	rtM50Ack				: R_TRIG;
	rtM61Ack				: R_TRIG;
	rtM62Ack				: R_TRIG;
	rtM63Ack				: R_TRIG;
	rtM64Ack				: R_TRIG;
	rtM65Ack				: R_TRIG;
	
	F_Ploter: FB_MX2;
	ui_PPodCzestotliwosc: INT;
	b_FP_CCW: BOOL;
	b_FP_CW: BOOL;
	b_FP_Reset: BOOL;
	seq:INT;
	czas:ARRAY[0..100] OF ton;
	R_Pobranie_Kierownica:R_TRIG;

	Zabral: BOOL;
	
	
	
	bZabral: BOOL;
	iStateRunning: INT;
	bServiceMove: BOOL;

END_VAR

VAR CONSTANT
	nAxes	 : WORD:=2;
END_VAR

// Always clear command in active step

// Read input signals
Act_InUpdate();

// ====================================================
// FBs CALL
Act_FBsCall();
// Monitoring
Act_Monitoring();
	
// Error collection
Act_Error();

Act_MovePath(); 

//automat plotera
A_Ploter_Auto();

// SAFETY CALL 
// Tylko komenda Abort dostepna jest niezaleznie od stanu
IF eMachineCommand = E_MachineCommand.eAbort AND eMachineState <> E_MachineState.eAborted THEN
	eMachineState := E_MachineState.eAborting;
END_IF

// Machine mode change over
CASE eMachineMode OF
	
	E_MachineMode.eAutomatic:
		Act_ModeAutomatic();
		
	E_MachineMode.eManual:
		Act_ModeManual();	
		
	E_MachineMode.eMaintenance:
		Act_ModeMaintenance();	
		
END_CASE

// Call Axis online FBs


// Write outputs
Act_OutUpdate(); 
A_FPloter();
A_Prawidlo();

(*//jogi
IF  GVL_HMI.bAuto=FALSE  THEN
	GVL_GLOBAL.bPlotJogF:=GVL_HMI.bHmiPlotCw;
	GVL_GLOBAL.bPlotJogB:=GVL_HMI.bHmiPlotCCw;
END_IF*)

ACTION A_FPloter:
F_Ploter
	(w_Status:=GVL_Omron.wOmron_Pl_Status,
	ui_CzestotliwoscI:=ui_PPodCzestotliwosc,
	b_CCW									:= b_FP_CCW, 
	b_CW									:= b_FP_CW,
	b_Reset                                 := b_FP_Reset,
	w_ControlW                              => GVL_Omron.wOmron_Pl_Control,
 	ui_CzestotliwoscO                       => GVL_Omron.iOmron_Pl_SeVelo,
);

	
	IF GVL_HMI.A_Start=TRUE AND GVL_HMI.bAuto=TRUE AND GVL_HMI.bEnablePloter=TRUE THEN 
		
	ui_PPodCzestotliwosc					:= 2500;
	b_FP_CCW								:= TRUE;		
	
	END_IF	
	IF GVL_HMI.A_Stop=TRUE OR GVL_HMI.bEnablePloter=FALSE THEN  

	b_FP_CCW								:= FALSE;		
	b_FP_CW:=FALSE;
	END_IF
	
	IF GVL_HMI.bAuto=FALSE AND GVL_GLOBAL.falownik_rolek_cewka=TRUE THEN 
	ui_PPodCzestotliwosc					:= 2500;	
	b_FP_CCW								:= TRUE;
	b_FP_CW 								:= FALSE;
	
	
	ELSIF GVL_HMI.bAuto=FALSE AND GVL_GLOBAL.falownik_pasow_cewka=FALSE THEN
	
	ui_PPodCzestotliwosc					:= 0;	
	b_FP_CCW								:= 0;
	b_FP_CW									:= 0;

	END_IF
END_ACTION

ACTION A_Ploter_Auto:
//prędkości osi 
					rItemPickVelocity:=GVL_Recipe.Predk_plot_ruch; 	//[mm/min]
					rItemPlaceVelocity:=GVL_Recipe.Predk_plot_ruch;	//[mm/min]
					rMoveVelocity:=GVL_Recipe.Predk_plot_pobranie;		//[mm/min]
//podglad bitów do obsłgui programu
					R_Pobranie_Kierownica(CLK:=GVL_GLOBAL.Zabierz_Z_Kierownicy);
					R_bReadyForMove(CLK:=bReadyForMove);
				
					bZabral;
					GVL_GLOBAL.odloz_do_kartonu;
//automat do plotera 
				(*	IF GVL_HMI.A_Stop=TRUE OR GVL_HMI.bEnablePloter=FALSE THEN	
					seq									:=0;
					END_IF
				*)	
//rozpoczęcie case
		CASE seq OF 
			0:(*start*)			
					IF GVL_HMI.A_Start=TRUE AND GVL_HMI.bEnablePloter=TRUE THEN	
					seq									:=2;
					END_IF
			2:(*Jazda do home i sprawdzenie stanów *)
					bReferneceHbot						:=TRUE;
					GVL_GLOBAL.zaw_chwyt1_auto			:=FALSE;
					GVL_GLOBAL.zaw_chwyt2_auto			:=FALSE;
					IF GVL_Machine.eState=60 AND bReadyForMove=TRUE AND rMoveMode=3  THEN 
					seq									:=3;
					END_IF
			3:(**)	
					IF bReadyForMove=TRUE AND czas[1].Q=TRUE THEN	
					bMoveCmd							:=TRUE;
					END_IF
					IF bReadyForMove=FALSE THEN	
					bMoveCmd							:=FALSE;
					seq									:=5;
					END_IF
			5:(*sprawdza czy dojechał jak dojechał to jedzie dalej *)
					IF bHome=TRUE THEN
					bHomeDone							:=TRUE;
					seq									:=7;
					END_IF			
			7:(*czeka az zniknie bit bhome*)		
					IF bHome=FALSE THEN
					bHomeDone							:=FALSE;
					seq									:=10;
					END_IF	
			10:(*jade pick pozycje*)
					
					bPickAndPlace						:=TRUE;
					IF rMoveMode=1 AND czas[2].Q=TRUE  THEN
					bPickAndPlace						:=FALSE;
					seq									:=13;
					END_IF
			13:(**)
					IF   bReadyForMove=TRUE THEN
					bMoveCmd							:=TRUE;
					seq									:=14;
					END_IF
			14:(**)	
					IF   bReadyForMove=FALSE THEN
					bMoveCmd							:=FALSE;
					seq									:=15;
					END_IF
			15:(**)	
					IF bReadyToPick=TRUE AND GVL_GLOBAL.Zabierz_Z_Kierownicy  THEN
					bReadyToPickACK						:=TRUE;
					seq									:=17;
					END_IF
			17:(**)	
					IF bReadyToPick=FALSE THEN
					bReadyToPickACK						:=FALSE;
					seq									:=19;						
					END_IF
			19:(**)
				 	IF bPicked=TRUE AND bZabral=TRUE THEN
					GVL_GLOBAL.zaw_chwyt1_auto			:=TRUE;
					GVL_GLOBAL.zaw_chwyt2_auto			:=TRUE;
					seq									:=20;	
					END_IF
					
			20:(*jedzio pobrac jak ma zgode*)

					IF bPicked=TRUE AND czas[4].Q=TRUE THEN
					bPickedACK							:=TRUE;						
					seq									:=22;
					END_IF
			22:(**)		
					IF bPicked=FALSE THEN
					bPickedACK							:=FALSE;						
					seq									:=25;
					END_IF			

					
			25:(*jak zgoda odklada*)
					IF bReadyToPlace=TRUE AND GVL_GLOBAL.odloz_do_kartonu=TRUE THEN
					bReadyToPlaceACK					:=TRUE;
					seq									:=27;
					END_IF

			27:(**)
					IF bReadyToPlace=FALSE   THEN
					bReadyToPlaceACK					:=FALSE;
					seq									:=30;
					END_IF
			30:(*potwierdzenie ze dojechal do pobrania *)
					IF bPlaced	=TRUE  THEN
					GVL_GLOBAL.Ploter_pobral			:=TRUE;
					bPlacedACK							:=TRUE;
					seq									:=33;
					END_IF
			33:(**)		
					IF bPlaced	=FALSE  THEN
					bPlacedACK							:=FALSE;
					seq									:=35;
					END_IF
			35:(*jak zgoda to jedzie spowrotem do pobrania *)
					GVL_GLOBAL.zaw_chwyt1_auto			:=FALSE;
					GVL_GLOBAL.zaw_chwyt2_auto			:=FALSE;
					bReturnToPick						:=TRUE;
					IF rMoveMode = 2  AND czas[3].Q=TRUE  THEN
					seq									:=40;
					END_IF
			40:(**)
					IF bReadyForMove=TRUE THEN
					bMoveCmd							:=TRUE;
					seq									:=43;	
					END_IF
			43:(**)
					IF bReadyForMove=FALSE THEN
					bMoveCmd							:=FALSE;
					seq									:=45;	
					END_IF

			45:(**)
					IF P_HBot_v3.stMcAxisOnline_MCS_X.stStatus.lrActPos<700 THEN 
					GVL_GLOBAL.bZaladowanyPrawidlo		:=TRUE;
					END_IF
					IF bPicked	=TRUE THEN	
					bPickedACK							:=TRUE;
					seq									:=50;//bedzie wracal do 10 
					END_IF
			50:(**)
					IF bPicked	=FALSE THEN	
					bPickedACK							:=FALSE;
					seq									:=10;//bedzie wracal do 10 					
					END_IF
			END_CASE
			czas[1](IN:=seq=3,PT:=T#1200MS);
			czas[2](IN:=rMoveMode=1,PT:=T#1200MS);
			czas[3](IN:=rMoveMode=2,PT:=T#1200MS);
			czas[4](IN:=seq=20,PT:=T#500MS);
			czas[9](IN:=bReferneceHbot,PT:=T#300MS);
			czas[12](IN:=GVL_GLOBAL.bZaladowanyPrawidlo,PT:=T#500MS);

			IF czas[12].Q=TRUE THEN
				GVL_GLOBAL.bZaladowanyPrawidlo	:=FALSE;
			END_IF
END_ACTION

ACTION A_Prawidlo:
FB_Prawidlo(
	b_Start:=GVL_HMI.A_Start AND GVL_HMI.bEnablePloter , 
	b_Stop:=GVL_HMI.A_Stop , 
	bKon_Hamulec1:=GVL_IO_P.b1B1 , 
	bKon_Hamulec2:=GVL_IO_P.b5B1 , 
	bKonPodajnik1:=GVL_IO_P.b6B1 , 
	bKonPodajnik2:=GVL_IO_P.b2B1 , 
	bCzHamulec:=GVL_IO_P.b3B1 , 
	bZaladowany:=GVL_GLOBAL.bZaladowanyPrawidlo	 , 
	bZaworPodnosnik1=>GVL_GLOBAL.zaw_prawidlo_auto , 
	bZaworPodnosnik2=>GVL_GLOBAL.zaw_prawidlo_dol_auto , 
	bZaworHamulec=>GVL_GLOBAL.zaw_hamulec_auto , 
	bZgodaNaRuch=>GVL_GLOBAL.bZgodaNaRuchPrawidlo , 
	bLaduj=>GVL_GLOBAL.odloz_do_kartonu );
END_ACTION

ACTION Act_Error:
// Program summary error
bError := 	tonAxesError.Q OR 
			PLCMachineMode[GVL_NCI.nChan].Error OR  
			PRG_KinTrans.eKinStatus = KinStatus_Error;
			// ie. Init Error
			// OR axis error
			// OR item error
END_ACTION

ACTION Act_FBsCall:

PRG_ChannelHandler();
fbMcAxisOnline_MCS_X(stMcAxisOnline:= stMcAxisOnline_MCS_X , Axis:= Axis_MCS_X);
fbMcAxisOnline_MCS_Y(stMcAxisOnline:= stMcAxisOnline_MCS_y , Axis:= Axis_MCS_Y);
fbMcAxisOnline_ACS_X(stMcAxisOnline:= stMcAxisOnline_ACS_X , Axis:= Axis_ACS_X);
fbMcAxisOnline_ACS_Y(stMcAxisOnline:= stMcAxisOnline_ACS_Y , Axis:= Axis_ACS_Y);	


//________Kinematic____________//
PRG_KinTrans(
	bBuildKinGroup:= , 
	bCleanKinGroup:= , 
	bResetKinGroup:= , 
	bKinBusy=> , 
	bKinDone=> , 
	bKinBuilt=> , 
	bKinClined=> , 
	bKinError=> , 
	udiKinErrorID=> , 
	eKinStatus=> );
//_____________________________//

//________NCI__________________//
PRG_GroupAxesToNci(	stMachineMode := PLCMachineMode[PLCSelectedChannel], 
					stAxisRef_X:= Axis_MCS_X, 
					stAxisRef_Y:= Axis_MCS_Y );

//_____________________________//
END_ACTION

ACTION Act_InUpdate:
bIn1 := TRUE; // Assign, filters, conditions, scaling etc
PLCMachineMode[GVL_NCI.nChan].ProgramName := 'C:\TwinCat\CNC\NC_1.nc';
END_ACTION

ACTION Act_ModeAutomatic:
// State Machine
CASE eMachineState OF

	E_MachineState.eIdle:
		
	
		// ====================================================
		// There should be main code
		// i.e. CASE iStepInit OF	
		// ====================================================
		// Allow for stop only if conditions are true - in this step we can wait without an error

		
		IF TRUE (* condition *) THEN
			eMachineState 						:= E_MachineState.eStopped;
		END_IF
		
		IF bError THEN
			eMachineState 						:= E_MachineState.eError;
		END_IF
		
	E_MachineState.eStopping:
		PLCMachineMode[GVL_NCI.nChan].Start:= FALSE;
		
		CASE iStateStoping OF
			0:
				PLCMachineMode[GVL_NCI.nChan].Stop:= TRUE;
				IF stMcAxisOnline_MCS_X.stStatus.stAxisStatus.NotMoving AND stMcAxisOnline_MCS_Y.stStatus.stAxisStatus.NotMoving THEN
					PLCMachineMode[GVL_NCI.nChan].Stop:= FALSE;
					iStateStoping := iStateStoping + 10;
				ELSIF stMcAxisOnline_MCS_X.stStatus.bNcError OR stMcAxisOnline_MCS_Y.stStatus.bNcError THEN
					iStateStoping := iStateStoping + 20;
				END_IF
			10:
				IF PRG_KinTrans.bKinBuilt THEN
					PRG_KinTrans.bCleanKinGroup := TRUE;
					iStateStoping := iStateStoping + 10;
				ELSE
					iStateStoping := iStateStoping + 20;	
				END_IF
			20:
				IF PRG_KinTrans.bKinDone THEN
					PRG_KinTrans.bCleanKinGroup 		:= FALSE;
					iStateStoping := iStateStoping + 10;
				ELSIF PRG_KinTrans.bKinError THEN
					PRG_KinTrans.bCleanKinGroup 		:= FALSE;
					iStateStoping := iStateStoping + 10;
				END_IF
				
			30:
				PLCMachineMode[GVL_NCI.nChan].Reset:= TRUE;
				IF ItpGetStateInterpreter(arrNCToPLC_NCIChannel_REF[1]) = 1 THEN
					PLCMachineMode[GVL_NCI.nChan].Reset := FALSE;
					iStateStoping := iStateStoping + 10;
				END_IF
			END_CASE
		IF iStateStoping = 40 (* condition *) THEN
			eMachineState 						:= E_MachineState.eStopped;
			iStateStoping 						:= 0;
		END_IF		
	
	E_MachineState.eStopped:
		
		stMcAxisOnline_MCS_X.mcPower.bEnable 			:= FALSE;
		stMcAxisOnline_MCS_X.mcPower.bEnable_Negative 	:= FALSE;
		stMcAxisOnline_MCS_X.mcPower.bEnable_Positive 	:= FALSE;

		stMcAxisOnline_MCS_Y.mcPower.bEnable 			:= FALSE;
		stMcAxisOnline_MCS_Y.mcPower.bEnable_Negative 	:= FALSE;
		stMcAxisOnline_MCS_Y.mcPower.bEnable_Positive 	:= FALSE;
		
		stMcAxisOnline_ACS_X.mcPower.bEnable 			:= FALSE;
		stMcAxisOnline_ACS_X.mcPower.bEnable_Negative 	:= FALSE;
		stMcAxisOnline_ACS_X.mcPower.bEnable_Positive 	:= FALSE;
		
		stMcAxisOnline_ACS_Y.mcPower.bEnable 			:= FALSE;
		stMcAxisOnline_ACS_Y.mcPower.bEnable_Negative 	:= FALSE;
		stMcAxisOnline_ACS_Y.mcPower.bEnable_Positive 	:= FALSE;
	
		
		IF eMachineCommand = E_MachineCommand.eRun THEN
			eMachineState 						:= E_MachineState.eStarting;
		END_IF

		IF eMachineCommand = E_MachineCommand.eRestart THEN
			GVL_Machine.eCommand				:= E_MachineCommand.eStop;
			eMachineState 						:= E_MachineState.eRestarting;
		END_IF			
				
		IF bError THEN
			eMachineState 						:= E_MachineState.eError;
		END_IF

	E_MachineState.eStarting:
		PLCMachineMode[GVL_NCI.nChan].Manual 	:= FALSE;

		CASE iStepStarting OF
			0:
				PLCMachineMode[GVL_NCI.nChan].Stop				:= FALSE;
				
				stMcAxisOnline_MCS_X.mcPower.bEnable 			:= TRUE;
				stMcAxisOnline_MCS_X.mcPower.bEnable_Negative 	:= TRUE;
				stMcAxisOnline_MCS_X.mcPower.bEnable_Positive 	:= TRUE;
				stMcAxisOnline_MCS_X.mcPower.lrOverride		 	:= 100.0;	
	
				stMcAxisOnline_MCS_Y.mcPower.bEnable 			:= TRUE;
				stMcAxisOnline_MCS_Y.mcPower.bEnable_Negative 	:= TRUE;
				stMcAxisOnline_MCS_Y.mcPower.bEnable_Positive 	:= TRUE;
				stMcAxisOnline_MCS_Y.mcPower.lrOverride		 	:= 100.0;	
				
				stMcAxisOnline_ACS_X.mcPower.bEnable 			:= TRUE;
				stMcAxisOnline_ACS_X.mcPower.bEnable_Negative 	:= TRUE;
				stMcAxisOnline_ACS_X.mcPower.bEnable_Positive 	:= TRUE;
				stMcAxisOnline_ACS_X.mcPower.lrOverride		 	:= 100.0;	
				
				stMcAxisOnline_ACS_Y.mcPower.bEnable 			:= TRUE;
				stMcAxisOnline_ACS_Y.mcPower.bEnable_Negative 	:= TRUE;
				stMcAxisOnline_ACS_Y.mcPower.bEnable_Positive 	:= TRUE;
				stMcAxisOnline_ACS_Y.mcPower.lrOverride		 	:= 100.0;	
				
				IF tonAxesReady.Q THEN
					iStepStarting := iStepStarting + 10;
				ELSIF tonAxesError.Q THEN
					bError := TRUE;
				END_IF
			10:
				PLCMachineMode[GVL_NCI.nChan].Automatic := TRUE;
				IF PLCNciChannelState.Mode[GVL_NCI.nChan] = 2 THEN
					iStepStarting := iStepStarting + 10;
				END_IF
			20:
			
				IF PRG_KinTrans.bKinBuilt AND NOT PRG_KinTrans.bKinError THEN
					iStepStarting := iStepStarting + 20;		
				ELSE
					iStepStarting := iStepStarting + 10;
				END_IF
				
			30:
				PRG_KinTrans.bBuildKinGroup := TRUE;
					IF PRG_KinTrans.bKinDone THEN
						PRG_KinTrans.bBuildKinGroup := FALSE;
						iStepStarting := iStepStarting + 10;
					END_IF
			40:
				;
			END_CASE 
	
		IF iStepStarting = 40 AND PRG_KinTrans.eKinStatus = KinStatus_Ready(* condition *) THEN
			eMachineState 						:= E_MachineState.eRunning;
			iStepStarting 						:= 0;
		END_IF
		
	E_MachineState.eRunning:
		
		//Act_MovePath();  do usuniecia
		PLCMachineMode[GVL_NCI.nChan].Start 	:= GVL_Machine.bNciStart;
		PLCMachineMode[GVL_NCI.nChan].Stop 		:= GVL_Machine.bNCiStop;
	
		GVL_Machine.bNciFeedHold := ItpIsEStopEx(arrNCToPLC_NCIChannel_REF[1]);
		
		// ====================================================
		// There should be main code
		// i.e. CASE iStepAuto OF
		// ====================================================
		IF eMachineCommand = E_MachineCommand.eStop OR bError THEN
			eMachineState 						:= E_MachineState.eStopping;
		END_IF

	E_MachineState.eAborting:

		// Stop and reset everything - usually SAFETY function
		CASE iStateAborting OF
			0:
				IF ItpGetStateInterpreter(arrNCToPLC_NCIChannel_REF[1]) <> 1 THEN
					iStateAborting := iStateAborting +10;
				ELSE
					iStateAborting := iStateAborting + 20;
				END_IF
			10:
				PLCMachineMode[GVL_NCI.nChan].Stop:= TRUE;
					IF ItpIsEStopEx(arrNCToPLC_NCIChannel_REF[1]) THEN
						PLCMachineMode[GVL_NCI.nChan].Stop:= FALSE;
						iStateAborting := iStateAborting +10;
					ELSIF 	ItpGetStateInterpreter(arrNCToPLC_NCIChannel_REF[1]) <> 1 OR
							ItpGetStateInterpreter(arrNCToPLC_NCIChannel_REF[1]) <> 12 OR
							ItpGetStateInterpreter(arrNCToPLC_NCIChannel_REF[1]) <> 13 THEN
						PLCMachineMode[GVL_NCI.nChan].Stop:= FALSE;
						iStateAborting := iStateAborting +10;
					END_IF
			20:
				IF PRG_KinTrans.bKinBuilt THEN
					PRG_KinTrans.bCleanKinGroup := TRUE;
					iStateAborting := iStateAborting + 10;
				ELSE	
					iStateAborting := iStateAborting + 20;
				END_IF
			30:
				IF PRG_KinTrans.bKinDone THEN
					PRG_KinTrans.bCleanKinGroup := FALSE;
					iStateAborting := iStateAborting + 10;
				ELSIF PRG_KinTrans.bKinError THEN
					PRG_KinTrans.bCleanKinGroup := FALSE;
					iStateAborting := iStateAborting + 10;
				END_IF
			40:	
				PLCMachineMode[GVL_NCI.nChan].Manual := TRUE;
				stMcAxisOnline_ACS_X.mcSS1.bExecute := TRUE;
				stMcAxisOnline_ACS_Y.mcSS1.bExecute := TRUE;
				IF stMcAxisOnline_ACS_X.mcSS1.bDone AND stMcAxisOnline_ACS_Y.mcSS1.bDone THEN
					iStateAborting := iStateAborting + 10;
				ELSIF stMcAxisOnline_ACS_X.mcSS1.bError OR stMcAxisOnline_ACS_Y.mcSS1.bError THEN
					iStateAborting := iStateAborting + 10;
				END_IF
			50:	

				stMcAxisOnline_MCS_X.mcSS1.bExecute := Axis_MCS_X.Status.PTPmode;
				stMcAxisOnline_MCS_Y.mcSS1.bExecute := Axis_MCS_Y.Status.PTPmode;
			
				IF 	stMcAxisOnline_MCS_X.mcSS1.bDone AND stMcAxisOnline_MCS_Y.mcSS1.bDone THEN
					iStateAborting := iStateAborting + 10;
				ELSIF stMcAxisOnline_MCS_X.mcSS1.bError OR stMcAxisOnline_MCS_Y.mcSS1.bError THEN
					iStateAborting := iStateAborting + 10;
				END_IF	
			
			60:
				stMcAxisOnline_MCS_X.mcSS1.bExecute := TRUE;
				stMcAxisOnline_MCS_Y.mcSS1.bExecute := TRUE;
				stMcAxisOnline_ACS_X.mcSS1.bExecute := TRUE;;
				stMcAxisOnline_ACS_Y.mcSS1.bExecute := TRUE;
		END_CASE
	
		IF iStateAborting = 60 THEN
			eMachineState 						:= E_MachineState.eAborted;
			iStateAborting						:= 0;
		END_IF		
		
	E_MachineState.eAborted:

		stMcAxisOnline_MCS_X.mcSS1.bExecute := NOT GVL_SafetyFrom_RT2.bSAFETY_PermissionSS1;
		stMcAxisOnline_MCS_Y.mcSS1.bExecute := NOT GVL_SafetyFrom_RT2.bSAFETY_PermissionSS1;
		stMcAxisOnline_ACS_X.mcSS1.bExecute := NOT GVL_SafetyFrom_RT2.bSAFETY_PermissionSS1;
		stMcAxisOnline_ACS_Y.mcSS1.bExecute := NOT GVL_SafetyFrom_RT2.bSAFETY_PermissionSS1;
					
		IF eMachineCommand = E_MachineCommand.eReset THEN
			eMachineState 						:= E_MachineState.eReseting;
		END_IF
		
		IF bError THEN
			eMachineState 						:= E_MachineState.eError;
		END_IF

	E_MachineState.eError:

		// ====================================================
		// Two types of error:
		// 1. 'Small/soft' Error - fix a problem and go to stop
		// 2. 'Serious/hard' Error - there is a need of restart everything, if there is a sequence - reset it too - fix a problem and go to init
		// ====================================================
		stMcAxisOnline_MCS_X.mcReset.bExecute	:= FALSE;	
		stMcAxisOnline_MCS_Y.mcReset.bExecute 	:= FALSE;	
		stMcAxisOnline_ACS_X.mcReset.bExecute 	:= FALSE;	
		stMcAxisOnline_ACS_Y.mcReset.bExecute 	:= FALSE;	
		stMcAxisOnline_MCS_X.mcStop.bExecute 	:= FALSE;
		stMcAxisOnline_MCS_Y.mcStop.bExecute	:= FALSE;
		stMcAxisOnline_ACS_X.mcStop.bExecute 	:= FALSE;
		stMcAxisOnline_ACS_Y.mcStop.bExecute	:= FALSE;
		PRG_KinTrans.bResetKinGroup 			:= FALSE;
		PRG_KinTrans.bBuildKinGroup 			:= FALSE;
		PRG_KinTrans.bCleanKinGroup 			:= FALSE;		
		PLCMachineMode[GVL_NCI.nChan].Reset 	:= FALSE;		
		PLCMachineMode[GVL_NCI.nChan].Stop		:= FALSE;
		PLCMachineMode[GVL_NCI.nChan].Start		:= FALSE;
	
		IF eMachineCommand = E_MachineCommand.eReset THEN
			eMachineState 						:= E_MachineState.eReseting;
		END_IF
		
		IF eMachineCommand = E_MachineCommand.eRestart THEN
			eMachineState 						:= E_MachineState.eRestarting;
		END_IF

	E_MachineState.eReseting:

		// ====================================================
		//'Small/soft' Error - fix a problem and go to stop
		// Reset drives only when it is necessary
		// ====================================================
		// Check if axis errors cleared
	
		IF PRG_KinTrans.eKinStatus = KinStatus_Error OR PRG_KinTrans.bKinError	THEN
			PRG_KinTrans.bResetKinGroup := TRUE;
		ELSIF PLCMachineMode[GVL_NCI.nChan].Error THEN
			PLCMachineMode[GVL_NCI.nChan].Reset := TRUE;
		ELSIF stMcAxisOnline_MCS_X.stError.bError THEN
			stMcAxisOnline_MCS_X.mcReset.bExecute := TRUE;
		ELSIF stMcAxisOnline_MCS_Y.stError.bError THEN
			stMcAxisOnline_MCS_Y.mcReset.bExecute := TRUE;	
		ELSIF stMcAxisOnline_ACS_X.stError.bError THEN
			stMcAxisOnline_ACS_X.mcReset.bExecute := TRUE;
		ELSIF stMcAxisOnline_ACS_Y.stError.bError THEN
			stMcAxisOnline_ACS_Y.mcReset.bExecute := TRUE;
		END_IF

	
		IF NOT tonAxesError.Q AND NOT PLCMachineMode[GVL_NCI.nChan].Error AND PRG_KinTrans.eKinStatus <> KinStatus_Error AND NOT PRG_KinTrans.bKinError THEN
			stMcAxisOnline_MCS_X.mcReset.bExecute	:= FALSE;	
			stMcAxisOnline_MCS_Y.mcReset.bExecute 	:= FALSE;	
			stMcAxisOnline_ACS_X.mcReset.bExecute 	:= FALSE;	
			stMcAxisOnline_ACS_Y.mcReset.bExecute 	:= FALSE;	
			PRG_KinTrans.bResetKinGroup 			:= FALSE;
			PLCMachineMode[GVL_NCI.nChan].Reset		:= FALSE;
			eMachineState  						:= E_MachineState.eStopping;
		END_IF
				
		// Blad bloku resetowania lub zakonczylismy kasowanie bledu osi, ale os jest nadal w bledzie, np. nie usunieta usterka - idz do kroku bledu
		IF bError (*(stAxis.stAxisDiagOutputs.Error OR (stAxis.stAxisDiagOutputs.Done AND stAxis.bAxisError)) *) THEN
			eMachineState  						:= E_MachineState.eError;
		END_IF
		
	E_MachineState.eRestarting:

		// ====================================================
		// 'Serious/hard' Error - there is a need of restart everything, if there is a sequence - reset it too - fix a problem and go to init
		// Reset drives only when it is necessary
		// ====================================================
		// Check if axis errors cleared
		bError := FALSE;
		
		IF TRUE (*NOT bAxisError AND NOT other errors *) THEN
			eMachineState  						:= E_MachineState.eIdle;
		END_IF
				
		// Blad bloku resetowania lub zakonczylismy kasowanie bledu osi, ale os jest nadal w bledzie, np. nie usunieta usterka - idz do kroku bledu
		IF bError (*(stAxis.stAxisDiagOutputs.Error OR (stAxis.stAxisDiagOutputs.Done AND stAxis.bAxisError)) *) THEN
			eMachineState  						:= E_MachineState.eError;
		END_IF
		
END_CASE
END_ACTION

ACTION Act_ModeMaintenance:
// State Machine
CASE eMachineState OF

	E_MachineState.eIdle, E_MachineState.eStopping, E_MachineState.eStopped, E_MachineState.eStarting:
	
		// ====================================================
		// There should be main code
		// i.e. CASE iStepInit OF	
		// ====================================================
		// Allow for stop only if conditions are true - in this step we can wait without an error	
		IF TRUE (* condition *) AND eMachineCommand = E_MachineCommand.eRun THEN
			eMachineState 						:= E_MachineState.eRunning;
		END_IF

	E_MachineState.eRunning:

		// ====================================================
		// HMI control
		// There should be main code,
		// i.e. CASE iStepAuto OF
		// ====================================================
		IF eMachineCommand = E_MachineCommand.eStop THEN
			eMachineState 						:= E_MachineState.eStopping;
		END_IF

	E_MachineState.eAborting:

		// Stop and reset everything - usually SAFETY function
		IF TRUE (* condition *) THEN
			eMachineState 						:= E_MachineState.eAborted;
		END_IF
		
	E_MachineState.eAborted:

		IF eMachineCommand = E_MachineCommand.eReset THEN
			eMachineState 						:= E_MachineState.eReseting;
		END_IF

	E_MachineState.eRestarting, E_MachineState.eReseting, E_MachineState.eError:

			;// Unused

END_CASE
END_ACTION

ACTION Act_ModeManual:
// State Machine

CASE eMachineState OF

	E_MachineState.eIdle:
	
		// ====================================================
		// There should be main code
		// i.e. CASE iStepInit OF	
		// ====================================================
		// Allow for stop only if conditions are true - in this step we can wait without an error

		CASE iStateIdle OF
			0:	//Wyłączenie kanału interpolacji
				PLCMachineMode[GVL_NCI.nChan].Automatic 		:= FALSE;
				PLCMachineMode[GVL_NCI.nChan].Manual			:= TRUE;
				IF arrNCToPLC_NCIChannel_REF[1].ItpState = 1 THEN
					iStateIdle := iStateIdle + 10;
				END_IF
			10:	
				IF PRG_KinTrans.bKinBuilt THEN
					PRG_KinTrans.bCleanKinGroup := TRUE;
					iStateIdle := iStateIdle + 10;
				ELSE
					iStateIdle := iStateIdle + 20;	
				END_IF
			20:
				IF PRG_KinTrans.bKinDone THEN
					PRG_KinTrans.bCleanKinGroup 		:= FALSE;
					iStateIdle := iStateIdle + 10;
				ELSIF PRG_KinTrans.bKinError THEN
					PRG_KinTrans.bCleanKinGroup 		:= FALSE;
					iStateIdle := iStateIdle + 10;
				END_IF
			END_CASE
	
		IF iStateIdle = 30 (* condition *)THEN
			eMachineState 						:= E_MachineState.eStopped;
			iStateIdle							:= 0;		
		END_IF
		
		IF bError THEN
			eMachineState 						:= E_MachineState.eError;
			iStateIdle							:= 0;	
		END_IF

	E_MachineState.eStopping:	
		CASE iStateStoping OF
			0:	

				stMcAxisOnline_MCS_X.mcStop.bExecute := TRUE;
				stMcAxisOnline_MCS_Y.mcStop.bExecute := TRUE;
				IF 	stMcAxisOnline_MCS_X.mcStop.bDone AND stMcAxisOnline_MCS_Y.mcStop.bDone THEN
					iStateStoping := iStateStoping + 10;
				ELSIF stMcAxisOnline_MCS_X.mcStop.bError OR stMcAxisOnline_MCS_Y.mcStop.bError THEN
					iStateStoping := iStateStoping + 10;
				END_IF	
			10:
				stMcAxisOnline_MCS_X.mcStop.bExecute := FALSE;
				stMcAxisOnline_MCS_Y.mcStop.bExecute := FALSE;
				iStateStoping := iStateStoping + 10;
			20:
				PRG_KinTrans.bCleanKinGroup := TRUE;
				IF PRG_KinTrans.bKinDone THEN
					PRG_KinTrans.bCleanKinGroup 		:= FALSE;
					iStateStoping := iStateStoping + 10;
				END_IF	
		END_CASE
		
		IF iStateStoping = 30 (* condition *) THEN
			eMachineState 						:= E_MachineState.eStopped;
			iStateStoping 						:= 0;
		END_IF			
	
		IF bError THEN
			eMachineState 						:= E_MachineState.eError;
		END_IF		
	
	E_MachineState.eStopped:
			
				stMcAxisOnline_MCS_X.mcPower.bEnable 			:= FALSE;
				stMcAxisOnline_MCS_X.mcPower.bEnable_Negative 	:= FALSE;
				stMcAxisOnline_MCS_X.mcPower.bEnable_Positive 	:= FALSE;
		
				stMcAxisOnline_MCS_Y.mcPower.bEnable 			:= FALSE;
				stMcAxisOnline_MCS_Y.mcPower.bEnable_Negative 	:= FALSE;
				stMcAxisOnline_MCS_Y.mcPower.bEnable_Positive 	:= FALSE;
				
				stMcAxisOnline_ACS_X.mcPower.bEnable 			:= FALSE;
				stMcAxisOnline_ACS_X.mcPower.bEnable_Negative 	:= FALSE;
				stMcAxisOnline_ACS_X.mcPower.bEnable_Positive 	:= FALSE;
				
				stMcAxisOnline_ACS_Y.mcPower.bEnable 			:= FALSE;
				stMcAxisOnline_ACS_Y.mcPower.bEnable_Negative 	:= FALSE;
				stMcAxisOnline_ACS_Y.mcPower.bEnable_Positive 	:= FALSE;
		IF eMachineCommand = E_MachineCommand.eRun THEN
			eMachineState 						:= E_MachineState.eStarting;
		END_IF	

		IF eMachineCommand = E_MachineCommand.eRestart THEN
			GVL_Machine.eCommand				:= E_MachineCommand.eStop;
			eMachineState 						:= E_MachineState.eRestarting;
		END_IF			
		
 	E_MachineState.eStarting:
		CASE iStepStarting OF
			0:
				stMcAxisOnline_MCS_X.mcPower.bEnable 			:= TRUE;
				stMcAxisOnline_MCS_X.mcPower.bEnable_Negative 	:= TRUE;
				stMcAxisOnline_MCS_X.mcPower.bEnable_Positive 	:= TRUE;
				stMcAxisOnline_MCS_X.mcPower.lrOverride		 	:= 100.0;	
			
				stMcAxisOnline_MCS_Y.mcPower.bEnable 			:= TRUE;
				stMcAxisOnline_MCS_Y.mcPower.bEnable_Negative 	:= TRUE;
				stMcAxisOnline_MCS_Y.mcPower.bEnable_Positive 	:= TRUE;
				stMcAxisOnline_MCS_Y.mcPower.lrOverride		 	:= 100.0;	
				
				stMcAxisOnline_ACS_X.mcPower.bEnable 			:= TRUE;
				stMcAxisOnline_ACS_X.mcPower.bEnable_Negative 	:= TRUE;
				stMcAxisOnline_ACS_X.mcPower.bEnable_Positive 	:= TRUE;
				stMcAxisOnline_ACS_X.mcPower.lrOverride		 	:= 100.0;	
				
				stMcAxisOnline_ACS_Y.mcPower.bEnable 			:= TRUE;
				stMcAxisOnline_ACS_Y.mcPower.bEnable_Negative 	:= TRUE;
				stMcAxisOnline_ACS_Y.mcPower.bEnable_Positive 	:= TRUE;
				stMcAxisOnline_ACS_Y.mcPower.lrOverride		 	:= 100.0;	
				IF tonAxesReady.Q THEN
					iStepStarting := iStepStarting + 10;
				END_IF
			10:
				IF PRG_KinTrans.bKinBuilt THEN
					iStepStarting := iStepStarting + 20;
				ELSE
					PRG_KinTrans.bBuildKinGroup := TRUE;
					iStepStarting := iStepStarting + 10;
				END_IF

			20:	
				IF PRG_KinTrans.bKinDone THEN
					PRG_KinTrans.bBuildKinGroup := FALSE;	
					iStepStarting := iStepStarting + 10;
				END_IF
			30:
				;	
		END_CASE
	
		IF iStepStarting = 30 THEN
			eMachineState 						:= E_MachineState.eRunning;
			iStepStarting 						:= 0;
		END_IF
				

		
		IF bError THEN
			eMachineState 							:= E_MachineState.eError;		
			iStepStarting							:= 0;			
		END_IF
	
		
		
	E_MachineState.eRunning:

		// ====================================================
		// HMI control
		// There should be main code,
		// i.e. CASE iStepAuto OF
		// ====================================================
		CASE iStateRunning OF
			0:
				stMcAxisOnline_MCS_Y.mcMoveAbsolute.bExecute := FALSE;
				stMcAxisOnline_MCS_X.mcMoveAbsolute.bExecute := FALSE;
				IF bServiceMove THEN
					bServiceMove := FALSE;
					iStateRunning := iStateRunning + 10;
				END_IF
			10:
				stMcAxisOnline_MCS_Y.mcMoveAbsolute.lrPosition :=  0; //Pozycja
				stMcAxisOnline_MCS_Y.mcMoveAbsolute.lrVelocity :=  10;      //Predkosc
				stMcAxisOnline_MCS_Y.mcMoveAbsolute.bExecute := TRUE;
				IF stMcAxisOnline_MCS_Y.mcMoveAbsolute.bDone THEN
					stMcAxisOnline_MCS_Y.mcMoveAbsolute.bExecute := FALSE;
					iStateRunning := iStateRunning + 10;
				END_IF
			20:
				
				stMcAxisOnline_MCS_X.mcMoveAbsolute.lrPosition :=  0; //Pozycja
				stMcAxisOnline_MCS_X.mcMoveAbsolute.lrVelocity :=  10;      //Predkosc
				stMcAxisOnline_MCS_X.mcMoveAbsolute.bExecute := TRUE;
				IF stMcAxisOnline_MCS_X.mcMoveAbsolute.bDone THEN
					stMcAxisOnline_MCS_X.mcMoveAbsolute.bExecute := FALSE;
					iStateRunning := iStateRunning + 10;
				END_IF
			30:
				;//Dummy wait
			
		END_CASE
		IF eMachineCommand = E_MachineCommand.eStop OR bError THEN
			eMachineState 						:= E_MachineState.eStopping;
			iStateRunning := 0;
		END_IF

	E_MachineState.eAborting:
		CASE iStateAborting OF
			0:
				PLCMachineMode[GVL_NCI.nChan].Automatic 		:= FALSE;
				PLCMachineMode[GVL_NCI.nChan].Manual	 		:= TRUE;
				iStateAborting := iStateAborting + 10;
			10:
				IF PRG_KinTrans.bKinBuilt THEN
					PRG_KinTrans.bCleanKinGroup := TRUE;
					iStateAborting := iStateAborting + 10;
				ELSE	
					iStateAborting := iStateAborting + 20;
				END_IF
			20:
				IF PRG_KinTrans.bKinDone THEN
					PRG_KinTrans.bCleanKinGroup := FALSE;
					iStateAborting := iStateAborting + 10;
				ELSIF PRG_KinTrans.bKinError THEN
					PRG_KinTrans.bCleanKinGroup := FALSE;
					iStateAborting := iStateAborting + 10;
				END_IF
			30:
				stMcAxisOnline_ACS_X.mcSS1.bExecute := TRUE;
				stMcAxisOnline_ACS_Y.mcSS1.bExecute := TRUE;
				
				IF stMcAxisOnline_ACS_X.mcSS1.bDone AND stMcAxisOnline_ACS_Y.mcSS1.bDone THEN
					iStateAborting := iStateAborting + 10;
				ELSIF stMcAxisOnline_ACS_X.mcSS1.bError OR stMcAxisOnline_ACS_Y.mcSS1.bError THEN
					iStateAborting := iStateAborting + 10;
				END_IF	
			40:
				stMcAxisOnline_MCS_X.mcSS1.bExecute := Axis_MCS_X.Status.PTPmode;
				stMcAxisOnline_MCS_Y.mcSS1.bExecute := Axis_MCS_Y.Status.PTPmode;
				IF 	stMcAxisOnline_MCS_X.mcSS1.bDone AND stMcAxisOnline_MCS_Y.mcSS1.bDone THEN
					iStateAborting := iStateAborting + 10;
				ELSIF stMcAxisOnline_MCS_X.mcSS1.bError OR stMcAxisOnline_MCS_Y.mcSS1.bError THEN
					iStateAborting := iStateAborting + 10;
				END_IF	
			50:
				stMcAxisOnline_MCS_X.mcSS1.bExecute := TRUE;
				stMcAxisOnline_MCS_Y.mcSS1.bExecute := TRUE;
				stMcAxisOnline_ACS_X.mcSS1.bExecute := TRUE;
				stMcAxisOnline_ACS_Y.mcSS1.bExecute := TRUE;
				eMachineState 						:= E_MachineState.eAborted;	
		END_CASE
		// Stop and reset everything - usually SAFETY function
		IF iStateAborting = 50 (* condition *) THEN
			eMachineState 						:= E_MachineState.eAborted;
			iStateAborting := 0;
		END_IF
		
	E_MachineState.eAborted:
	
		stMcAxisOnline_MCS_X.mcSS1.bExecute := NOT GVL_SafetyFrom_RT2.bSAFETY_PermissionSS1;
		stMcAxisOnline_MCS_Y.mcSS1.bExecute := NOT GVL_SafetyFrom_RT2.bSAFETY_PermissionSS1;
		stMcAxisOnline_ACS_X.mcSS1.bExecute := NOT GVL_SafetyFrom_RT2.bSAFETY_PermissionSS1;
		stMcAxisOnline_ACS_Y.mcSS1.bExecute := NOT GVL_SafetyFrom_RT2.bSAFETY_PermissionSS1;
		IF eMachineCommand = E_MachineCommand.eReset THEN
			eMachineState 						:= E_MachineState.eReseting;
		END_IF

	E_MachineState.eError:

		// ====================================================
		// Two types of error:
		// 1. 'Small/soft' Error - fix a problem and go to stop
		// 2. 'Serious/hard' Error - there is a need of restart everything, if there is a sequence - reset it too - fix a problem and go to init
		// ====================================================
		stMcAxisOnline_MCS_X.mcReset.bExecute	:= FALSE;	
		stMcAxisOnline_MCS_Y.mcReset.bExecute 	:= FALSE;	
		stMcAxisOnline_ACS_X.mcReset.bExecute 	:= FALSE;	
		stMcAxisOnline_ACS_Y.mcReset.bExecute 	:= FALSE;	
		stMcAxisOnline_MCS_X.mcStop.bExecute 	:= FALSE;
		stMcAxisOnline_MCS_Y.mcStop.bExecute	:= FALSE;
		stMcAxisOnline_ACS_X.mcStop.bExecute 	:= FALSE;
		stMcAxisOnline_ACS_Y.mcStop.bExecute	:= FALSE;
		PRG_KinTrans.bResetKinGroup 			:= FALSE;
		PRG_KinTrans.bBuildKinGroup 			:= FALSE;	
		PRG_KinTrans.bCleanKinGroup 			:= FALSE;		
	
		IF eMachineCommand = E_MachineCommand.eReset THEN
			eMachineState 						:= E_MachineState.eReseting;
		END_IF
		
		IF eMachineCommand = E_MachineCommand.eRestart THEN
			eMachineState 						:= E_MachineState.eRestarting;
		END_IF		
			
		
	E_MachineState.eRestarting, E_MachineState.eReseting:
	
		IF PRG_KinTrans.eKinStatus = KinStatus_Error	THEN
			PRG_KinTrans.bResetKinGroup := TRUE;
		ELSIF PLCMachineMode[GVL_NCI.nChan].Error THEN
			PLCMachineMode[GVL_NCI.nChan].Reset := TRUE;
		ELSIF stMcAxisOnline_MCS_X.stError.bError THEN
			stMcAxisOnline_MCS_X.mcReset.bExecute := TRUE;
		ELSIF stMcAxisOnline_MCS_Y.stError.bError THEN
			stMcAxisOnline_MCS_Y.mcReset.bExecute := TRUE;	
		ELSIF stMcAxisOnline_ACS_X.stError.bError THEN
			stMcAxisOnline_ACS_X.mcReset.bExecute := TRUE;
		ELSIF stMcAxisOnline_ACS_Y.stError.bError THEN
			stMcAxisOnline_ACS_Y.mcReset.bExecute := TRUE;
		END_IF	
	
		IF NOT tonAxesError.Q AND NOT PLCMachineMode[GVL_NCI.nChan].Error AND PRG_KinTrans.eKinStatus <> KinStatus_Error THEN
			stMcAxisOnline_MCS_X.mcReset.bExecute	:= FALSE;	
			stMcAxisOnline_MCS_Y.mcReset.bExecute 	:= FALSE;	
			stMcAxisOnline_ACS_X.mcReset.bExecute 	:= FALSE;	
			stMcAxisOnline_ACS_Y.mcReset.bExecute 	:= FALSE;	
			PRG_KinTrans.bResetKinGroup 			:= FALSE;
			PLCMachineMode[GVL_NCI.nChan].Reset		:= FALSE;
			
			IF eMachineState = E_MachineState.eReseting THEN
				eMachineState  						:= E_MachineState.eStopping;
			END_IF
			
			IF eMachineState = E_MachineState.eRestarting THEN
				eMachineState  						:= E_MachineState.eIdle;	
			END_IF
		END_IF	
	(*
		// Blad bloku resetowania lub zakonczylismy kasowanie bledu osi, ale os jest nadal w bledzie, np. nie usunieta usterka - idz do kroku bledu
		IF bError (*(stAxis.stAxisDiagOutputs.Error OR (stAxis.stAxisDiagOutputs.Done AND stAxis.bAxisError)) *) THEN
			eMachineState  						:= E_MachineState.eError;
		END_IF
			;// Unused
	*)
END_CASE
END_ACTION

ACTION Act_Monitoring:
// Ustawianie flag, monitoring kolizjii, watchdogi, jazdy po krzywce itp
tonAxesReady.IN := 	stMcAxisOnline_ACS_X.mcPower.bStatus AND stMcAxisOnline_ACS_X.stStatus.bAxisReady AND
					stMcAxisOnline_ACS_Y.mcPower.bStatus AND stMcAxisOnline_ACS_Y.stStatus.bAxisReady AND
					stMcAxisOnline_MCS_X.mcPower.bStatus AND stMcAxisOnline_MCS_X.stStatus.bAxisReady AND
					stMcAxisOnline_MCS_Y.mcPower.bStatus AND stMcAxisOnline_MCS_Y.stStatus.bAxisReady	;
tonAxesReady(PT:=T#200MS);

tonAxesError.IN := 	stMcAxisOnline_ACS_X.stError.bDriveError OR stMcAxisOnline_ACS_X.stError.bNcError OR
					stMcAxisOnline_ACS_Y.stError.bDriveError OR stMcAxisOnline_ACS_Y.stError.bNcError OR
					stMcAxisOnline_MCS_X.stError.bDriveError OR stMcAxisOnline_MCS_X.stError.bNcError OR
					stMcAxisOnline_MCS_Y.stError.bDriveError OR stMcAxisOnline_MCS_Y.stError.bNcError	;
tonAxesError(PT:=T#200MS);
END_ACTION

ACTION Act_MovePath:
nRParamWrite[1,10] := rMoveMode;				//[mm]
nRParamWrite[1,11] := rPickItemHigh;			//[mm]
nRParamWrite[1,12] := rPlaceItemHigh;			//[mm/min]
nRParamWrite[1,13] := 60 * rItemPickVelocity; 	//[mm/min]
nRParamWrite[1,14] := 60 * rItemPlaceVelocity;	//[mm/min]
nRParamWrite[1,15] := 60 * rMoveVelocity;		//[mm/min]

bReadyForMove		:= bMFunc[1,50];
bReadyToPick 		:= bMFunc[1,61]; 	// Item Picked
bPicked		 		:= bMFunc[1,62]; 	// Item Picked
bReadyToPlace 		:= bMFunc[1,63];	// ItemP laced
bPlaced		 		:= bMFunc[1,64];	// ItemP laced
bHome				:= bMFunc[1,65];

rtM50Ack(CLK:= bMoveCmd			);
rtM61Ack(CLK:= bReadyToPickACK	);
rtM62Ack(CLK:= bPickedACK		);
rtM63Ack(CLK:= bReadyToPlaceACK	);
rtM64Ack(CLK:= bPlacedACK		);
rtM65Ack(CLK:= bHomeDone		);

bQuitMFunc[1,50] 	:= rtM50Ack.Q;
bQuitMFunc[1,61] 	:= rtM61Ack.Q;
bQuitMFunc[1,62] 	:= rtM62Ack.Q;
bQuitMFunc[1,63] 	:= rtM63Ack.Q;
bQuitMFunc[1,64] 	:= rtM64Ack.Q;
bQuitMFunc[1,65] 	:= rtM65Ack.Q;

// Mode selector
IF bPickAndPlace THEN
	bPickAndPlace	:= FALSE;
	bReturnToPick 	:= FALSE;	
	bReferneceHbot 	:= FALSE;
	rMoveMode 		:= 1;
END_IF

IF bReturnToPick AND NOT bPickAndPlace AND NOT bReferneceHbot THEN
	bReturnToPick 	:= FALSE;
	bPickAndPlace 	:= FALSE;	
	bReferneceHbot	:= FALSE;	
	rMoveMode 		:= 2;
END_IF

IF bReferneceHbot AND NOT bPickAndPlace AND NOT bReturnToPick THEN
	bReferneceHbot	:= FALSE;	
	bPickAndPlace 	:= FALSE;	
	bReturnToPick 	:= FALSE;	
	rMoveMode 		:= 3;
END_IF
//_________________________________________________
END_ACTION

ACTION Act_OutUpdate:
;
END_ACTION

END_PROGRAM

// ---- POUs/Programy/Hbot/AxisOnline/POUsAxisOnline/AX5000/FB_McAxisOnlineAX5000.TcPOU
(*
//==================================================================================================
//							Beckhoff Automation Poland
//									23.05.2018
//	Wszystkomajacy blok funkcyjny do sterowania osia, 
//	wymagane biblioteki: Tc2_EtherCAT, Tc2_Drive, Tc2_MC2_Drive, Tc2_MC2, Tc2_Utilities
// 	v1.0 	|| TC v 3.1.4022.16	 	|| - first edition
//==================================================================================================
Do zmiany
*)
FUNCTION_BLOCK FB_McAxisOnlineAX5000

VAR_IN_OUT
	stMcAxisOnline						: ST_McAxisOnline;
	Axis								: AXIS_REF;
END_VAR
VAR
	mcPower								: MC_Power;
	mcStop								: MC_Stop;
	mcHalt								: MC_Halt;
	mcStopSS1							: MC_Stop;
	mcStopSS2							: MC_Stop;
	mcReset								: MC_Reset;
	mcHome								: MC_Home;
	mcSetPosition						: MC_SetPosition;
	fbSetPositionOffset					: FB_SetPositionOffset;
	mcJog								: MC_Jog;

	mcMoveAbsolute						: MC_MoveAbsolute;
	mcMoveRelative						: MC_MoveRelative;
	mcMoveVelocity						: MC_MoveVelocity;
	mcMoveModulo						: MC_MoveModulo;
	mcMoveAbsolute2						: MC_MoveAbsolute;
	mcMoveRelative2						: MC_MoveRelative;
	mcMoveVelocity2						: MC_MoveVelocity;
	mcMoveModulo2						: MC_MoveModulo;

	fbMotorMonitoring					: FB_MotorMonitoringAX5000;
	fbHoldingBrakeCtrl					: FB_HoldingBrakeCtrlAX5000;
	fbNcLimitSwitch						: FB_NcSWLimitSwitchCtrl;
	tonGetDriveDiag						: TON;
	fbReadChannelErrorCode				: FB_AxisDiag;
	
	mcReadDriveAddress					: MC_ReadDriveAddress;
	mcReadParameterSet					: MC_ReadParameterSet;
	fbGetDriveRef						: FB_GetDriveRef;

	// Internal
	bInitialized						: BOOL;
			
// Initialization
	iInitStep							: INT;
	bInitializationError				: BOOL;
	wInitializationErrorCounter			: WORD;
	bDriveAddressReady					: BOOL;
	bDriveRefReady						: BOOL;
	bReadParameterSetReady				: BOOL;
	tonDelay							: TON;
// Re init
	udiOnlineChangeCntOld				: UDINT;
	bOnlineChangeDetected				: BOOL;
	bReInit								: BOOL;
	bReInitialized						: BOOL;
	bReInitializationError				: BOOL;
	// Axis diag struct
	stAX5000Diag						: ST_AX5000Diag;
	{attribute 'instance-path'}
	{attribute 'noinit'}
	sInstancePath						: STRING;
END_VAR

// Device dependent initialization 
ACT_Initialization();
// Device independent commands, mostly NC 
ACT_States();
ACT_SWLimitSwitch();
ACT_Stop();
ACT_Power();
ACT_Homing();
ACT_Jog();
ACT_Move();
ACT_ResetAndDiag();
ACT_SetPosition();
// Device dependent commands
// Motor monitoring possible only with real axis
IF NOT Axis.Status.OpMode.SimulationAxis THEN
	ACT_MotorMonitoring();
END_IF
// Device dependent commands, possible only on real axis after complete initialization
IF bInitialized AND NOT Axis.Status.OpMode.SimulationAxis THEN
	ACT_SetPositionIO();
	ACT_HoldingBrakeCtrl();
END_IF

// Device independent error collection
ACT_ErrorCollection();

ACTION ACT_ErrorCollection:
// Error flags
stMcAxisOnline.stError.bDriveError					:= Axis.Status.DriveDeviceError;

stMcAxisOnline.stError.bNcError						:= Axis.Status.Error;

stMcAxisOnline.stError.bFBError						:= stMcAxisOnline.mcPower.bError OR stMcAxisOnline.mcReset.bError OR stMcAxisOnline.mcHome.bError OR stMcAxisOnline.mcJog.bError
													OR stMcAxisOnline.mcHalt.bError OR stMcAxisOnline.mcStop.bError OR stMcAxisOnline.mcSS1.bError OR stMcAxisOnline.mcSS2.bError
													OR stMcAxisOnline.mcMoveAbsolute.bError OR stMcAxisOnline.mcMoveRelative.bError OR stMcAxisOnline.mcMoveVelocity.bError OR stMcAxisOnline.mcMoveModulo.bError
													OR stMcAxisOnline.mcMoveAbsolute2.bError OR stMcAxisOnline.mcMoveRelative2.bError OR stMcAxisOnline.mcMoveVelocity2.bError OR stMcAxisOnline.mcMoveModulo2.bError
													OR stMcAxisOnline.stNcLimitSwitch.bError OR stMcAxisOnline.mcSetPosition.bError;
									
stMcAxisOnline.stError.bCommunicationError			:= stMcAxisOnline.stChannelErrorCode.bError OR stMcAxisOnline.stSetPositionOffset.bError OR stMcAxisOnline.stMotorMonitoring.bError OR stMcAxisOnline.stHoldingBrake.bError;

stMcAxisOnline.stError.bError						:= stMcAxisOnline.stError.bDriveError OR stMcAxisOnline.stError.bNcError OR stMcAxisOnline.stError.bFBError OR stMcAxisOnline.stError.bCommunicationError;
stMcAxisOnline.bError								:= stMcAxisOnline.stError.bError; // Forward one stage up

// Error codes
stMcAxisOnline.stError.uiDriveErrorID 				:= stMcAxisOnline.stChannelErrorCode.uiChannelErrorCode;
stMcAxisOnline.stError.uiDriveErrorIDHex 			:= stMcAxisOnline.stChannelErrorCode.uiChannelErrorCodeHex;

stMcAxisOnline.stError.udiNcErrorID 				:= Axis.Status.ErrorID;
stMcAxisOnline.stError.udiNcErrorIDHex 				:= Axis.Status.ErrorID;
	

stMcAxisOnline.stError.udiFBErrorID 				:= 	stMcAxisOnline.mcPower.udiErrorID + 
														stMcAxisOnline.mcReset.udiErrorID + 
														stMcAxisOnline.mcHome.udiErrorID + 
														stMcAxisOnline.mcJog.udiErrorID +
														stMcAxisOnline.mcHalt.udiErrorID + 
														stMcAxisOnline.mcStop.udiErrorID + 
														stMcAxisOnline.mcSS1.udiErrorID + 
														stMcAxisOnline.mcSS2.udiErrorID +
														stMcAxisOnline.mcMoveAbsolute.udiErrorID + 
														stMcAxisOnline.mcMoveRelative.udiErrorID + 
														stMcAxisOnline.mcMoveVelocity.udiErrorID + 
														stMcAxisOnline.mcMoveModulo.udiErrorID +
														stMcAxisOnline.mcMoveAbsolute2.udiErrorID + 
														stMcAxisOnline.mcMoveRelative2.udiErrorID + 
														stMcAxisOnline.mcMoveVelocity2.udiErrorID + 
														stMcAxisOnline.mcMoveModulo2.udiErrorID +
														stMcAxisOnline.stNcLimitSwitch.udiErrorID + 
														stMcAxisOnline.mcSetPosition.udiErrorID;

stMcAxisOnline.stError.udiFBErrorIDHex 				:= stMcAxisOnline.stError.udiFBErrorID;

stMcAxisOnline.stError.udiErrorID					:= stMcAxisOnline.stSetPositionOffset.udiErrorID;
stMcAxisOnline.stError.uiAdsErrorID					:= stMcAxisOnline.stChannelErrorCode.uiAdsErrId + stMcAxisOnline.stMotorMonitoring.uiAdsErrId + stMcAxisOnline.stHoldingBrake.uiAdsErrId;
stMcAxisOnline.stError.uiSecErrorID					:= stMcAxisOnline.stChannelErrorCode.uiSecErrId + stMcAxisOnline.stMotorMonitoring.uiSecErrId + stMcAxisOnline.stHoldingBrake.uiSecErrId;
END_ACTION

ACTION ACT_HoldingBrakeCtrl:
fbHoldingBrakeCtrl(
					bForceLock			:= stMcAxisOnline.stHoldingBrake.bForceLock,
					bForceUnlock		:= stMcAxisOnline.stHoldingBrake.bForceUnlock,
					bBusy				=> stMcAxisOnline.stHoldingBrake.bBusy,
					bError				=> stMcAxisOnline.stHoldingBrake.bError,
					iAdsErrId			=> stMcAxisOnline.stHoldingBrake.uiAdsErrId,
					iSecErrId			=>stMcAxisOnline.stHoldingBrake.uiSecErrId , 
					Axis				:= Axis );
END_ACTION

ACTION ACT_Homing:
mcHome(		Axis						:= Axis,
			Execute						:= stMcAxisOnline.mcHome.bExecute,
			Position					:= stMcAxisOnline.mcHome.lrPosition,
			HomingMode					:= stMcAxisOnline.mcHome.eHomingMode,
			BufferMode					:= stMcAxisOnline.mcHome.eBufferMode,
			Options						:= stMcAxisOnline.mcHome.stOptions,
			bCalibrationCam				:= stMcAxisOnline.mcHome.bCalibrationCam,
			Done						=> stMcAxisOnline.mcHome.bDone,
			Busy						=> stMcAxisOnline.mcHome.bBusy,
			Active						=> stMcAxisOnline.mcHome.bActive,
			CommandAborted				=> stMcAxisOnline.mcHome.bCommandAborted,
			Error						=> stMcAxisOnline.mcHome.bError,
			ErrorID						=> stMcAxisOnline.mcHome.udiErrorID);
END_ACTION

ACTION ACT_Initialization:
// Init sequence of AX8000 drives. bInitialized flag is set just once. 
// bReInitialized ise set each time we do online change or request reinit operation
// bDriveAddressReady, bReadParameterSetReady, bDriveRefReady - set just once after successed read

// Online change detection
bOnlineChangeDetected					:= udiOnlineChangeCntOld <> _AppInfo.OnlineChangeCnt;
udiOnlineChangeCntOld 					:= _AppInfo.OnlineChangeCnt;
// Reset init
IF bReInit OR bOnlineChangeDetected THEN
	iInitStep							:= 0;
END_IF

//Initialization process
CASE iInitStep OF
	0:	// Read Drive Address
		
		stMcAxisOnline.mcReadDriveAddress.bExecute	:=	 TRUE;
		iInitStep						:= iInitStep + 10;
		
	10: // Wait for data
	
		IF NOT stMcAxisOnline.mcReadDriveAddress.bBusy THEN
			stMcAxisOnline.mcReadDriveAddress.bExecute	:=	 FALSE;
			IF stMcAxisOnline.mcReadDriveAddress.bDone THEN
				iInitStep 				:= iInitStep + 10;
				bDriveAddressReady 		:= TRUE;
			ELSE
				iInitStep 				:= 1000;		// Error step
			END_IF
		END_IF
		
	20:	// Read Parameter Set
		
		stMcAxisOnline.mcReadParameterSet.bExecute		:=	 TRUE;
		iInitStep						:= iInitStep + 10;
		
	30: // Wait for data
	
		IF NOT stMcAxisOnline.mcReadParameterSet.bBusy THEN
			stMcAxisOnline.mcReadParameterSet.bExecute	:=	 FALSE;
			IF stMcAxisOnline.mcReadParameterSet.bDone THEN
				iInitStep 				:= iInitStep + 10;
				bReadParameterSetReady 	:= TRUE;
			ELSE
				iInitStep 				:= 1000;		// Error step
			END_IF
		END_IF	
	
	40:	// Get Drive Ref
		
		stMcAxisOnline.stGetDriveRef.bExecute		:=	 TRUE;
		iInitStep						:= iInitStep + 10;
		
	50: // Wait for data
	
		IF NOT stMcAxisOnline.stGetDriveRef.bBusy THEN
			stMcAxisOnline.stGetDriveRef.bExecute	:=	 FALSE;
			IF NOT stMcAxisOnline.stGetDriveRef.bError THEN
				iInitStep 				:= iInitStep + 10;
				bDriveRefReady 			:= TRUE;
			ELSE
				iInitStep 				:= 1000;		// Error step
			END_IF
		END_IF
	
	60: // Success - initialized flag, clear error
		bReInitialized					:= bInitialized;	// TRUE only when it's not first initialization e.g. online change
		bInitialized 					:= TRUE;
		bReInitializationError			:= FALSE;			// TRUE only when it's not first initialization e.g. online change
		bInitializationError			:= FALSE;
		iInitStep 						:= iInitStep + 10;
		
	70: // Idle
	
		;
		
	1000: // Error step
		wInitializationErrorCounter 	:= wInitializationErrorCounter + 1;
		IF wInitializationErrorCounter < 100 THEN
			iInitStep					:= iInitStep + 5;			// Go to delay
		ELSE
			bReInitializationError		:= bInitializationError;	// TRUE only when it's not first initialization e.g. online change
			bInitializationError		:= TRUE;
			bReInitialized				:= FALSE;
			iInitStep 					:= iInitStep + 10;
		END_IF

	1005: // Delay step
		tonDelay(IN:= TRUE, PT:= T#1S);
		IF tonDelay.Q THEN
			tonDelay(IN:= FALSE, PT:= T#1S);
			iInitStep					:= 0;
		END_IF
		
	1010: // Idle after error
		;
	
END_CASE

mcReadDriveAddress(	Axis				:= Axis,
					Execute				:= stMcAxisOnline.mcReadDriveAddress.bExecute,
					Done				=> stMcAxisOnline.mcReadDriveAddress.bDone,
					Busy				=> stMcAxisOnline.mcReadDriveAddress.bBusy,
					Error				=> stMcAxisOnline.mcReadDriveAddress.bError,
					ErrorID				=> stMcAxisOnline.mcReadDriveAddress.udiErrorID,
					DriveAddress		=> stMcAxisOnline.stDriveAddress);
				
mcReadParameterSet(	Parameter			:= stMcAxisOnline.stAxisParameter,
					Axis				:= Axis,
					Execute				:= stMcAxisOnline.mcReadParameterSet.bExecute,
					Done				=> stMcAxisOnline.mcReadParameterSet.bDone,
					Busy				=> stMcAxisOnline.mcReadParameterSet.bBusy,
					Error				=> stMcAxisOnline.mcReadParameterSet.bError,
					ErrorID				=> stMcAxisOnline.mcReadParameterSet.udiErrorID);
					
fbGetDriveRef(		bExecute			:= stMcAxisOnline.stGetDriveRef.bExecute,
					bBusy				=> stMcAxisOnline.stGetDriveRef.bBusy,
					bError				=> stMcAxisOnline.stGetDriveRef.bError,
					udiErrorID			=> stMcAxisOnline.stGetDriveRef.udiErrorID,
					stDriveRef			=> stMcAxisOnline.stDriveRef,
					Axis				:= Axis);
END_ACTION

ACTION ACT_Jog:
// Direct access from bSlow or bFast, if none then free choice
IF stMcAxisOnline.mcJog.bSlowForward OR stMcAxisOnline.mcJog.bSlowBackward THEN
	stMcAxisOnline.mcJog.eMode			:= MC_JOGMODE_STANDARD_SLOW;
ELSIF stMcAxisOnline.mcJog.bFastForward OR stMcAxisOnline.mcJog.bFastBackward THEN
	stMcAxisOnline.mcJog.eMode			:= MC_JOGMODE_STANDARD_FAST;
END_IF

mcJog(		Axis						:= Axis,
			JogForward					:= stMcAxisOnline.mcJog.bJogForward OR stMcAxisOnline.mcJog.bSlowForward OR stMcAxisOnline.mcJog.bFastForward,
			JogBackwards				:= stMcAxisOnline.mcJog.bJogBackwards OR stMcAxisOnline.mcJog.bSlowBackward OR stMcAxisOnline.mcJog.bFastBackward,
			Mode						:= stMcAxisOnline.mcJog.eMode,
			Position					:= stMcAxisOnline.mcJog.lrPosition,
			Velocity					:= stMcAxisOnline.mcJog.lrVelocity,
			Acceleration				:= stMcAxisOnline.mcJog.lrAcceleration,
			Deceleration				:= stMcAxisOnline.mcJog.lrDeceleration,
			Jerk						:= stMcAxisOnline.mcJog.lrJerk,
			Done						=> stMcAxisOnline.mcJog.bDone,
			Busy						=> stMcAxisOnline.mcJog.bBusy,
			Active						=> stMcAxisOnline.mcJog.bActive,
			CommandAborted				=> stMcAxisOnline.mcJog.bCommandAborted,
			Error						=> stMcAxisOnline.mcJog.bError,
			ErrorID						=> stMcAxisOnline.mcJog.udiErrorID);
END_ACTION

ACTION ACT_MotorMonitoring:
fbMotorMonitoring(
					bReset				:= stMcAxisOnline.stMotorMonitoring.bReset, 
					rTorqueLimit		:= stMcAxisOnline.stMotorMonitoring.rTorqueLimit , 
					bError				=> stMcAxisOnline.stMotorMonitoring.bError , 
					iAdsErrId			=> stMcAxisOnline.stMotorMonitoring.uiAdsErrId , 
					iSercosErrId		=> stMcAxisOnline.stMotorMonitoring.uiSecErrId, 
					bInitialized		=> stMcAxisOnline.stMotorMonitoring.bInitialized , 
					bWarning			=> stMcAxisOnline.stMotorMonitoring.bWarning , 
					rWarningCurrent		=> stMcAxisOnline.stMotorMonitoring.rWarningCurrent , 
					rTorquePerc			=> stMcAxisOnline.stMotorMonitoring.rTorquePerc,
					rTorquePercMax		=> stMcAxisOnline.stMotorMonitoring.rTorquePercMax,
					rTorque				=> stMcAxisOnline.stMotorMonitoring.rTorque , 
					rTorqueF			=> stMcAxisOnline.stMotorMonitoring.rTorqueF , 
					rTorqueMax			=> stMcAxisOnline.stMotorMonitoring.rTorqueMax , 
					rCurrent			=> stMcAxisOnline.stMotorMonitoring.rCurrent , 
					rCurrentF			=> stMcAxisOnline.stMotorMonitoring.rCurrentF , 
					rCurrentMax			=> stMcAxisOnline.stMotorMonitoring.rCurrentMax , 
					rI2T				=> stMcAxisOnline.stMotorMonitoring.rI2T , 
					rI2TMax				=> stMcAxisOnline.stMotorMonitoring.rI2TMax , 
					Axis				:= Axis );
END_ACTION

ACTION ACT_Move:
{region "Primary"}
mcMoveAbsolute(	Axis					:= Axis,
				Execute					:= stMcAxisOnline.mcMoveAbsolute.bExecute,
				Position				:= stMcAxisOnline.mcMoveAbsolute.lrPosition,
				Velocity				:= stMcAxisOnline.mcMoveAbsolute.lrVelocity,
				Acceleration			:= stMcAxisOnline.mcMoveAbsolute.lrAcceleration,
				Deceleration			:= stMcAxisOnline.mcMoveAbsolute.lrDeceleration,
				Jerk					:= stMcAxisOnline.mcMoveAbsolute.lrJerk,
				BufferMode				:= stMcAxisOnline.mcMoveAbsolute.eBufferMode,
				Options					:= stMcAxisOnline.mcMoveAbsolute.stOptions,
				Done					=> stMcAxisOnline.mcMoveAbsolute.bDone,
				Busy					=> stMcAxisOnline.mcMoveAbsolute.bBusy,
				Active					=> stMcAxisOnline.mcMoveAbsolute.bActive,
				CommandAborted			=> stMcAxisOnline.mcMoveAbsolute.bCommandAborted,
				Error					=> stMcAxisOnline.mcMoveAbsolute.bError,
				ErrorID					=> stMcAxisOnline.mcMoveAbsolute.udiErrorID);

mcMoveRelative(	Axis					:= Axis,
				Execute					:= stMcAxisOnline.mcMoveRelative.bExecute,
				Distance				:= stMcAxisOnline.mcMoveRelative.lrDistance,
				Velocity				:= stMcAxisOnline.mcMoveRelative.lrVelocity,
				Acceleration			:= stMcAxisOnline.mcMoveRelative.lrAcceleration,
				Deceleration			:= stMcAxisOnline.mcMoveRelative.lrDeceleration,
				Jerk					:= stMcAxisOnline.mcMoveRelative.lrJerk,
				BufferMode				:= stMcAxisOnline.mcMoveRelative.eBufferMode,
				Options					:= stMcAxisOnline.mcMoveRelative.stOptions,
				Done					=> stMcAxisOnline.mcMoveRelative.bDone,
				Busy					=> stMcAxisOnline.mcMoveRelative.bBusy,
				Active					=> stMcAxisOnline.mcMoveRelative.bActive,
				CommandAborted			=> stMcAxisOnline.mcMoveRelative.bCommandAborted,
				Error					=> stMcAxisOnline.mcMoveRelative.bError,
				ErrorID					=> stMcAxisOnline.mcMoveRelative.udiErrorID);
				
mcMoveVelocity(	Axis					:= Axis,
				Execute					:= stMcAxisOnline.mcMoveVelocity.bExecute,
				Velocity				:= stMcAxisOnline.mcMoveVelocity.lrVelocity,
				Acceleration			:= stMcAxisOnline.mcMoveVelocity.lrAcceleration,
				Deceleration			:= stMcAxisOnline.mcMoveVelocity.lrDeceleration,
				Jerk					:= stMcAxisOnline.mcMoveVelocity.lrJerk,
				Direction				:= stMcAxisOnline.mcMoveVelocity.eDirection,
				BufferMode				:= stMcAxisOnline.mcMoveVelocity.eBufferMode,
				Options					:= stMcAxisOnline.mcMoveVelocity.stOptions,
				InVelocity				=> stMcAxisOnline.mcMoveVelocity.bInVelocity,
				Busy					=> stMcAxisOnline.mcMoveVelocity.bBusy,
				Active					=> stMcAxisOnline.mcMoveVelocity.bActive,
				CommandAborted			=> stMcAxisOnline.mcMoveVelocity.bCommandAborted,
				Error					=> stMcAxisOnline.mcMoveVelocity.bError,
				ErrorID					=> stMcAxisOnline.mcMoveVelocity.udiErrorID);
stMcAxisOnline.mcMoveVelocity.bDone		:= stMcAxisOnline.mcMoveVelocity.bInVelocity;

mcMoveModulo(	Axis					:= Axis,
				Execute					:= stMcAxisOnline.mcMoveModulo.bExecute,
				Position				:= stMcAxisOnline.mcMoveModulo.lrPosition,
				Velocity				:= stMcAxisOnline.mcMoveModulo.lrVelocity,
				Acceleration			:= stMcAxisOnline.mcMoveModulo.lrAcceleration,
				Deceleration			:= stMcAxisOnline.mcMoveModulo.lrDeceleration,
				Jerk					:= stMcAxisOnline.mcMoveModulo.lrJerk,
				Direction				:= stMcAxisOnline.mcMoveModulo.eDirection,
				BufferMode				:= stMcAxisOnline.mcMoveModulo.eBufferMode,
				Options					:= stMcAxisOnline.mcMoveModulo.stOptions,
				Done					=> stMcAxisOnline.mcMoveModulo.bDone,
				Busy					=> stMcAxisOnline.mcMoveModulo.bBusy,
				Active					=> stMcAxisOnline.mcMoveModulo.bActive,
				CommandAborted			=> stMcAxisOnline.mcMoveModulo.bCommandAborted,
				Error					=> stMcAxisOnline.mcMoveModulo.bError,
				ErrorID					=> stMcAxisOnline.mcMoveModulo.udiErrorID);
{endregion}
{region "Secondary"}
mcMoveAbsolute2(Axis					:= Axis,
				Execute					:= stMcAxisOnline.mcMoveAbsolute2.bExecute,
				Position				:= stMcAxisOnline.mcMoveAbsolute2.lrPosition,
				Velocity				:= stMcAxisOnline.mcMoveAbsolute2.lrVelocity,
				Acceleration			:= stMcAxisOnline.mcMoveAbsolute2.lrAcceleration,
				Deceleration			:= stMcAxisOnline.mcMoveAbsolute2.lrDeceleration,
				Jerk					:= stMcAxisOnline.mcMoveAbsolute2.lrJerk,
				BufferMode				:= stMcAxisOnline.mcMoveAbsolute2.eBufferMode,
				Options					:= stMcAxisOnline.mcMoveAbsolute2.stOptions,
				Done					=> stMcAxisOnline.mcMoveAbsolute2.bDone,
				Busy					=> stMcAxisOnline.mcMoveAbsolute2.bBusy,
				Active					=> stMcAxisOnline.mcMoveAbsolute2.bActive,
				CommandAborted			=> stMcAxisOnline.mcMoveAbsolute2.bCommandAborted,
				Error					=> stMcAxisOnline.mcMoveAbsolute2.bError,
				ErrorID					=> stMcAxisOnline.mcMoveAbsolute2.udiErrorID);

mcMoveRelative2(Axis					:= Axis,
				Execute					:= stMcAxisOnline.mcMoveRelative2.bExecute,
				Distance				:= stMcAxisOnline.mcMoveRelative2.lrDistance,
				Velocity				:= stMcAxisOnline.mcMoveRelative2.lrVelocity,
				Acceleration			:= stMcAxisOnline.mcMoveRelative2.lrAcceleration,
				Deceleration			:= stMcAxisOnline.mcMoveRelative2.lrDeceleration,
				Jerk					:= stMcAxisOnline.mcMoveRelative2.lrJerk,
				BufferMode				:= stMcAxisOnline.mcMoveRelative2.eBufferMode,
				Options					:= stMcAxisOnline.mcMoveRelative2.stOptions,
				Done					=> stMcAxisOnline.mcMoveRelative2.bDone,
				Busy					=> stMcAxisOnline.mcMoveRelative2.bBusy,
				Active					=> stMcAxisOnline.mcMoveRelative2.bActive,
				CommandAborted			=> stMcAxisOnline.mcMoveRelative2.bCommandAborted,
				Error					=> stMcAxisOnline.mcMoveRelative2.bError,
				ErrorID					=> stMcAxisOnline.mcMoveRelative2.udiErrorID);
				
mcMoveVelocity2(Axis					:= Axis,
				Execute					:= stMcAxisOnline.mcMoveVelocity2.bExecute,
				Velocity				:= stMcAxisOnline.mcMoveVelocity2.lrVelocity,
				Acceleration			:= stMcAxisOnline.mcMoveVelocity2.lrAcceleration,
				Deceleration			:= stMcAxisOnline.mcMoveVelocity2.lrDeceleration,
				Jerk					:= stMcAxisOnline.mcMoveVelocity2.lrJerk,
				Direction				:= stMcAxisOnline.mcMoveVelocity2.eDirection,
				BufferMode				:= stMcAxisOnline.mcMoveVelocity2.eBufferMode,
				Options					:= stMcAxisOnline.mcMoveVelocity2.stOptions,
				InVelocity				=> stMcAxisOnline.mcMoveVelocity2.bInVelocity,
				Busy					=> stMcAxisOnline.mcMoveVelocity2.bBusy,
				Active					=> stMcAxisOnline.mcMoveVelocity2.bActive,
				CommandAborted			=> stMcAxisOnline.mcMoveVelocity2.bCommandAborted,
				Error					=> stMcAxisOnline.mcMoveVelocity2.bError,
				ErrorID					=> stMcAxisOnline.mcMoveVelocity2.udiErrorID);
stMcAxisOnline.mcMoveVelocity2.bDone	:= stMcAxisOnline.mcMoveVelocity2.bInVelocity;

mcMoveModulo2(	Axis					:= Axis,
				Execute					:= stMcAxisOnline.mcMoveModulo2.bExecute,
				Position				:= stMcAxisOnline.mcMoveModulo2.lrPosition,
				Velocity				:= stMcAxisOnline.mcMoveModulo2.lrVelocity,
				Acceleration			:= stMcAxisOnline.mcMoveModulo2.lrAcceleration,
				Deceleration			:= stMcAxisOnline.mcMoveModulo2.lrDeceleration,
				Jerk					:= stMcAxisOnline.mcMoveModulo2.lrJerk,
				Direction				:= stMcAxisOnline.mcMoveModulo2.eDirection,
				BufferMode				:= stMcAxisOnline.mcMoveModulo2.eBufferMode,
				Options					:= stMcAxisOnline.mcMoveModulo2.stOptions,
				Done					=> stMcAxisOnline.mcMoveModulo2.bDone,
				Busy					=> stMcAxisOnline.mcMoveModulo2.bBusy,
				Active					=> stMcAxisOnline.mcMoveModulo2.bActive,
				CommandAborted			=> stMcAxisOnline.mcMoveModulo2.bCommandAborted,
				Error					=> stMcAxisOnline.mcMoveModulo2.bError,
				ErrorID					=> stMcAxisOnline.mcMoveModulo2.udiErrorID);
{endregion}
END_ACTION

ACTION ACT_Power:
mcPower(	Axis						:= Axis,									//
			Enable						:= stMcAxisOnline.mcPower.bEnable,
			Enable_Positive				:= stMcAxisOnline.mcPower.bEnable_Positive,
			Enable_Negative				:= stMcAxisOnline.mcPower.bEnable_Negative,
			Override					:= stMcAxisOnline.mcPower.lrOverride,
			BufferMode					:= stMcAxisOnline.mcPower.eBufferMode,
			Options						:= stMcAxisOnline.mcPower.stOptions,
			Status						=> stMcAxisOnline.mcPower.bStatus,
			Busy						=> stMcAxisOnline.mcPower.bBusy,
			Active						=> stMcAxisOnline.mcPower.bActive,
			Error						=> stMcAxisOnline.mcPower.bError,
			ErrorID						=> stMcAxisOnline.mcPower.udiErrorID);
END_ACTION

ACTION ACT_ResetAndDiag:
tonGetDriveDiag(IN:= stMcAxisOnline.stError.bDriveError AND NOT tonGetDriveDiag.Q, PT:= T#5S, Q=> , ET=> );

IF Axis.Status.OpMode.SimulationAxis THEN
	mcReset(
		Axis						:= Axis,
		Execute						:= stMcAxisOnline.mcReset.bExecute,
		Done						=> stMcAxisOnline.mcReset.bDone,
		Busy						=> stMcAxisOnline.mcReset.bBusy,
		Error						=> stMcAxisOnline.mcReset.bError,
		ErrorID						=> stMcAxisOnline.mcReset.udiErrorID);	
ELSE
	fbReadChannelErrorCode(
		Reset:=					stMcAxisOnline.mcReset.bExecute,
		GetDiag				:=	(stMcAxisOnline.stChannelErrorCode.bExecute OR tonGetDriveDiag.Q),
		Axis				:=	Axis , 
		stAX5000Diag		:=	stAX5000Diag , 
		Error				=> 	stMcAxisOnline.mcReset.bError , 
		AdsErrId			=>	stMcAxisOnline.mcReset.udiErrorID , 
		SercosErrId			=>	stMcAxisOnline.stChannelErrorCode.uiAdsErrId, //???
		ResetAct			=> , 
		DiagAct				=> , 
		Busy				=> 	stMcAxisOnline.mcReset.bBusy );
	
	stMcAxisOnline.stChannelErrorCode.bError 				:= stAX5000Diag.bC1DError;
	stMcAxisOnline.stChannelErrorCode.uiChannelErrorCode 	:= UDINT_TO_UINT (stAX5000Diag.iDiagNumber);
	stMcAxisOnline.stChannelErrorCode.uiChannelErrorCodeHex := UDINT_TO_UINT (stAX5000Diag.iDiagNumber);
END_IF
END_ACTION

ACTION ACT_SetPosition:
mcSetPosition(		Axis				:= Axis,
					Execute				:= stMcAxisOnline.mcSetPosition.bExecute,
					Position			:= stMcAxisOnline.mcSetPosition.lrPosition,
					Mode				:= stMcAxisOnline.mcSetPosition.bMode,
					Options				:= stMcAxisOnline.mcSetPosition.stOptions,
					Done				=> stMcAxisOnline.mcSetPosition.bDone,
					Busy				=> stMcAxisOnline.mcSetPosition.bBusy,
					Error				=> stMcAxisOnline.mcSetPosition.bError,
					ErrorID				=> stMcAxisOnline.mcSetPosition.udiErrorID);
END_ACTION

ACTION ACT_SetPositionIO:
fbSetPositionOffset(
	bExecute			:= stMcAxisOnline.stSetPositionOffset.bExecute , 
	lrPosition			:= stMcAxisOnline.stSetPositionOffset.lrPosition , 
	bRelative			:= stMcAxisOnline.stSetPositionOffset.bRelative , 
	eFeedback			:= stMcAxisOnline.stSetPositionOffset.eFeedback , 
	eMemory				:= stMcAxisOnline.stSetPositionOffset.eMemory , 
	bBusy				=> stMcAxisOnline.stSetPositionOffset.bBusy , 
	bError				=> stMcAxisOnline.stSetPositionOffset.bError, 
	udiErrorID			=> stMcAxisOnline.stSetPositionOffset.udiErrorID, 
	uiSoEErrorID		=> stMcAxisOnline.stSetPositionOffset.uiSecErrId,
	Axis				:= Axis );
END_ACTION

ACTION ACT_States:
// Read States and forward main states
Axis.ReadStatus();
stMcAxisOnline.stStatus.stAxisStatus		:= Axis.Status;
stMcAxisOnline.stStatus.dwAxisId			:= Axis.NcToPlc.AxisId;
stMcAxisOnline.stStatus.bNcError			:= Axis.Status.Error;
stMcAxisOnline.stStatus.udiNcErrorCode		:= Axis.Status.ErrorID;
stMcAxisOnline.stStatus.udiNcErrorCodeHex	:= Axis.Status.ErrorID;

stMcAxisOnline.stStatus.sAxisName			:= stMcAxisOnline.stAxisParameter.sAxisName;
stMcAxisOnline.stStatus.lrActPos			:= Axis.NcToPlc.ActPos;
stMcAxisOnline.stStatus.lrModuloActPos		:= Axis.NcToPlc.ModuloActPos;
stMcAxisOnline.stStatus.lrActVelo			:= Axis.NcToPlc.ActVelo;
stMcAxisOnline.stStatus.lrActAcc			:= Axis.NcToPlc.ActAcc;
stMcAxisOnline.stStatus.lrActTorque			:= Axis.NcToPlc.ActTorque;
stMcAxisOnline.stStatus.lrPosDiff			:= Axis.NcToPlc.PosDiff;
stMcAxisOnline.stStatus.lrSetPos			:= Axis.NcToPlc.SetPos;
stMcAxisOnline.stStatus.lrSetVelo			:= Axis.NcToPlc.SetVelo;
stMcAxisOnline.stStatus.lrSetAcc			:= Axis.NcToPlc.SetAcc;
stMcAxisOnline.stStatus.lrSetTorque			:= Axis.NcToPlc.SetTorque;
stMcAxisOnline.stStatus.lrPosDiff			:= Axis.NcToPlc.PosDiff;
stMcAxisOnline.stStatus.bAxisReady			:= Axis.Status.Operational;
stMcAxisOnline.stStatus.bHomed				:= Axis.Status.Homed;
stMcAxisOnline.stStatus.bCoupled			:= Axis.Status.Coupled;

// zezwolenie na zjazd z krancowki hw
Axis.PlcToNc.ControlDWord.8				:= stMcAxisOnline.stStatus.bAcceptBlockedDrive;
END_ACTION

ACTION ACT_Stop:
mcHalt(		Axis						:= Axis,
			Execute						:= stMcAxisOnline.mcHalt.bExecute,
			Deceleration				:= stMcAxisOnline.mcHalt.lrDeceleration,
			Jerk						:= stMcAxisOnline.mcHalt.lrJerk,
			BufferMode					:= stMcAxisOnline.mcHalt.eBufferMode,
			Options						:= stMcAxisOnline.mcHalt.stOptions,
			Done						=> stMcAxisOnline.mcHalt.bDone,
			Busy						=> stMcAxisOnline.mcHalt.bBusy,
			Active						=> stMcAxisOnline.mcHalt.bActive,
			CommandAborted				=> stMcAxisOnline.mcHalt.bCommandAborted,
			Error						=> stMcAxisOnline.mcHalt.bError,
			ErrorID						=> stMcAxisOnline.mcHalt.udiErrorID);
			
mcStop(		Axis						:= Axis,
			Execute						:= stMcAxisOnline.mcStop.bExecute,
			Deceleration				:= stMcAxisOnline.mcStop.lrDeceleration,
			Jerk						:= stMcAxisOnline.mcStop.lrJerk,
			Options						:= stMcAxisOnline.mcStop.stOptions,
			Done						=> stMcAxisOnline.mcStop.bDone,
			Busy						=> stMcAxisOnline.mcStop.bBusy,
			Active						=> stMcAxisOnline.mcStop.bActive,
			CommandAborted				=> stMcAxisOnline.mcStop.bCommandAborted,
			Error						=> stMcAxisOnline.mcStop.bError,
			ErrorID						=> stMcAxisOnline.mcStop.udiErrorID);
			
mcStopSS2(	Axis						:= Axis,
			Execute						:= stMcAxisOnline.mcSS2.bExecute,
			Deceleration				:= stMcAxisOnline.mcSS2.lrDeceleration,
			Jerk						:= stMcAxisOnline.mcSS2.lrJerk,
			Options						:= stMcAxisOnline.mcSS2.stOptions,
			Done						=> stMcAxisOnline.mcSS2.bDone,
			Busy						=> stMcAxisOnline.mcSS2.bBusy,
			Active						=> stMcAxisOnline.mcSS2.bActive,
			CommandAborted				=> stMcAxisOnline.mcSS2.bCommandAborted,
			Error						=> stMcAxisOnline.mcSS2.bError,
			ErrorID						=> stMcAxisOnline.mcSS2.udiErrorID);
			
mcStopSS1(	Axis						:= Axis,
			Execute						:= stMcAxisOnline.mcSS1.bExecute,
			Deceleration				:= stMcAxisOnline.mcSS1.lrDeceleration,
			Jerk						:= stMcAxisOnline.mcSS1.lrJerk,
			Options						:= stMcAxisOnline.mcSS1.stOptions,
			Done						=> stMcAxisOnline.mcSS1.bDone,
			Busy						=> stMcAxisOnline.mcSS1.bBusy,
			Active						=> stMcAxisOnline.mcSS1.bActive,
			CommandAborted				=> stMcAxisOnline.mcSS1.bCommandAborted,
			Error						=> stMcAxisOnline.mcSS1.bError,
			ErrorID						=> stMcAxisOnline.mcSS1.udiErrorID);
// SS1 - after MC_Stop function we have to disable drive			
stMcAxisOnline.mcPower.bEnable R= stMcAxisOnline.mcPower.bEnable_Positive R= stMcAxisOnline.mcPower.bEnable_Negative R= (stMcAxisOnline.mcSS1.bDone OR stMcAxisOnline.mcSS1.bCommandAborted OR stMcAxisOnline.mcSS1.bError);
END_ACTION

ACTION ACT_SWLimitSwitch:
fbNcLimitSwitch(	udiAxisID		:= Axis.NcToPlc.AxisId, 
					bRead			:= stMcAxisOnline.stNcLimitSwitch.bRead, 
					bWrite			:= stMcAxisOnline.stNcLimitSwitch.bWrite, 
					bReset			:= stMcAxisOnline.stNcLimitSwitch.bReset, 
					lrSetMinPos		:= stMcAxisOnline.stNcLimitSwitch.lrSetMinPos, 
					lrSetMaxPos		:= stMcAxisOnline.stNcLimitSwitch.lrSetMaxPos, 
					bSetMinMon		:= stMcAxisOnline.stNcLimitSwitch.bSetMinMon, 
					bSetMaxMon		:= stMcAxisOnline.stNcLimitSwitch.bSetMaxMon, 
					bBusy			=> stMcAxisOnline.stNcLimitSwitch.bBusy, 
					bError			=> stMcAxisOnline.stNcLimitSwitch.bError, 
					udiErrorID		=> stMcAxisOnline.stNcLimitSwitch.udiErrorID, 
					lrActMinPos		=> stMcAxisOnline.stNcLimitSwitch.lrActMinPos, 
					lrActMaxPos		=> stMcAxisOnline.stNcLimitSwitch.lrActMaxPos, 
					bActMinMon		=> stMcAxisOnline.stNcLimitSwitch.bActMinMon, 
					bActMaxMon		=> stMcAxisOnline.stNcLimitSwitch.bActMaxMon);
END_ACTION

END_FUNCTION_BLOCK

// ---- POUs/Programy/Hbot/AxisOnline/POUsAxisOnline/AX5000/FB_SetPositionOffset.TcPOU
//==================================================================================================
//							Beckhoff Automation Poland
//								23.05.2018
//	Blok do uzupełniania offsetu w enkoderze/AX5000
//	Obsluguje bledy zwiazane z wymiana silnika na nowy - bez wpisanego offsetu.
//	Naprawia błąd: 	0x0000F340- Position offset invalid.
//					0x0000F341- Position offset: No position offset excisting.
//	Aby wpisać wartość, silnik musi być wyłączony.
//	Niezbędne biblioteki:
//	Tc2_MC2;	Tc2_Utilities;	Tc2_MC2_Drive;	Tc2_EtherCAT, Tc2_Drive;
//
// 	v2.3	|| TC v 3.1.4022.16		|| - optymalizacja kodu
//	v2.2 	|| TC v 3.1.4022.2	 	|| - Poprawka w komentarzu
//	v2.1 	|| TC v 3.1.4022.0	 	|| - Uproszczono kod
//	v2.0 	|| TC v 3.1.4022.0	 	|| - Dodano obsługę AX52xx, przebudowano bloczek z wykorzystaniem FB_ChangeSlaveState
//	v1.0 	|| TC v 3.1.4020.32 	|| - Pierwsza wersja
//==================================================================================================
FUNCTION_BLOCK FB_SetPositionOffset
VAR_INPUT
	bExecute								: BOOL;							// rising edge starts sequence
	lrPosition								: LREAL		:=	0.001;			// Write new encoder position
	bRelative								: BOOL;							// When this flag is set, the position is relatively interpreted
	eFeedback								: E_PositionOffsetFeedback;		// ePositionOffsetFeedback1:= 0			ePositionOffsetFeedback2 := 1
	eMemory									: E_PositionOffsetMemory;		// ePositionOffsetMemory_Encoder:= 0	ePositionOffsetMemory_Drive := 1
END_VAR
VAR_OUTPUT
	bBusy									: BOOL;
	bError									: BOOL;	
	udiErrorID								: UDINT;						// bError=TRUE AND udiErrorID=0 means state request timeout
	uiSoEErrorID							: UINT;
END_VAR
VAR_IN_OUT
	Axis									: AXIS_REF;
END_VAR
VAR CONSTANT
	NCIDXG_AXPARMS							: UDINT			:= 16#4000;		// ADS group number to axis parameters 
	NCIDXO_AXP_HWAMSADDR					: UDINT			:= 16#31;		// ADS offset to drive channel
END_VAR
VAR
	rtExecute								: R_TRIG;						// bExecute triggers start
	fbSoEReset								: FB_SoEReset;
	fbSoEWritePassword						: FB_SoEWritePassword;			// unlock P-0-0278
	fbSoEAX5000SetPositionOffset			: FB_SoEAX5000SetPositionOffset;
	fbSoEReadDiagNumber						: FB_SoEReadDiagNumber;	
	fbSoEWrite_ByDriveRef					: FB_SoEWrite_ByDriveRef;
	fbSoERead_ByDriveRef					: FB_SoERead_ByDriveRef;
	fbChangeSlaveState						: FB_ChangeEtherCATSlaveState;
	fbAdsRead								: ADSREAD;
	stPlcDriveRef							: ST_PlcDriveRef;				// ADS buffer (need to change aNetId into sNetId)
	stDriveRef								: ST_DriveRef;					// come from stPlcDriveRef
	bDualChannel							: BOOL;
	stSoE_String							: ST_SoE_String;				// buffer for byDualChannel
	P_0_0278_Value							: WORD;							//	0- NO	1- YES
	iStep									: INT;							// Actual Step
	iLastStep								: INT;							// Last step before error
END_VAR

rtExecute	(CLK:= bExecute );

CASE iStep	OF

	0:																//	Enable FB, lock input parameters
		IF rtExecute.Q THEN
			bBusy							:= TRUE;
			bError							:= FALSE;
			udiErrorID						:= 0;
			uiSoEErrorID					:= 0;
			iLastStep						:= 0;
			fbSoEAX5000SetPositionOffset.Position := lrPosition; 
			fbSoEAX5000SetPositionOffset.Memory	:= eMemory;
			fbSoEAX5000SetPositionOffset.Relative := bRelative;
			fbSoEAX5000SetPositionOffset.Feedback := eFeedback;
			iStep							:= iStep + 10;
		END_IF			

	10:																// Get Drive channel from AXIS_REF by ADS
		fbAdsRead.NETID						:= '';
		fbAdsRead.PORT						:= AMSPORT_R0_NC;		// set ADS Port to NC
		fbAdsRead.IDXGRP					:= NCIDXG_AXPARMS + Axis.NcToPlc.AxisId;	// set ADS Group to AXIS Parameters
		fbAdsRead.IDXOFFS					:= NCIDXO_AXP_HWAMSADDR;// set ADS offset to channel number
		fbAdsRead.LEN						:= SIZEOF(stPlcDriveRef);
		fbAdsRead.DESTADDR					:= ADR(stPlcDriveRef);
		fbAdsRead.TMOUT						:= T#5S;
		fbAdsRead.READ						:= TRUE;
		iStep								:= iStep + 10;
		
	20:																// reading actual channel (DriveNo) from AXIS_REF	
		fbAdsRead.READ						:= FALSE;
		IF NOT fbAdsRead.BUSY AND NOT fbAdsRead.ERR THEN
			iStep							:= iStep + 10;	
			stDriveRef.sNetId				:= F_CreateAmsNetId(stPlcDriveRef.aNetId);	// change AmsNetId array into string
			stDriveRef.nSlaveAddr			:= stPlcDriveRef.nSlaveAddr;
			stDriveRef.nDriveNo				:= stPlcDriveRef.nDriveNo;	
			fbChangeSlaveState.sEtherCAT_NetID:= stDriveRef.sNetId;
			fbChangeSlaveState.nSlaveAddr	:= stDriveRef.nSlaveAddr;
		ELSIF fbAdsRead.ERR THEN
			udiErrorID						:= fbAdsRead.ERRID;
			iLastStep						:= iStep;
			iStep							:= 999;				
		END_IF
		
	30:																// Read drive diag number
		fbSoEReadDiagNumber.NetId			:= '';
		fbSoEReadDiagNumber.Execute			:= TRUE;
		iStep								:= iStep + 10;

	40:																// Choose method
		fbSoEReadDiagNumber.Execute			:= FALSE;
		IF NOT fbSoEReadDiagNumber.Busy THEN
			IF fbSoEReadDiagNumber.DiagNumber = (16#F341 OR 16#F340) THEN
				iStep						:= 50;					// Position errors -> Reset errors and write 
			ELSIF	fbSoEReadDiagNumber.DiagNumber >= (16#F000) THEN
				iLastStep					:= iStep;				// Do nothing in other error states
				iStep						:= 999;
			ELSE												
				iStep						:= 200;					// Drive Ready -> Write without changing OP State			
			END_IF
		END_IF
	
	50:																// Request INIT State
		fbChangeSlaveState.byReguestedState	:= EC_DEVICE_STATE_INIT;
		fbChangeSlaveState.bExecute			:= TRUE;
		iStep								:= iStep + 10;

	60,80:															// Wait till state changed
		fbChangeSlaveState.bExecute			:= FALSE;	
		IF NOT fbChangeSlaveState.bBusy AND NOT fbChangeSlaveState.bError THEN
			iStep							:= iStep + 10;
		ELSIF NOT fbChangeSlaveState.bBusy AND fbChangeSlaveState.bError THEN
			udiErrorID						:= fbChangeSlaveState.udiErrorID;
			iLastStep						:= iStep;
			iStep 							:= 999;
		END_IF
		
	70:																// Request PreOP State	
		fbChangeSlaveState.byReguestedState	:= EC_DEVICE_STATE_PREOP;
		fbChangeSlaveState.bExecute			:= TRUE;
		iStep								:= iStep + 10;
		
	90:																// Write drive password (unlock P-0-0278)
		fbSoEWritePassword.Password.strData	:= 'AX5000';
		fbSoEWritePassword.NetId			:= '';
		fbSoEWritePassword.Execute			:= TRUE;
		iStep								:= iStep + 10;
		
	100:															// wait till password passes
		fbSoEWritePassword.Execute			:= FALSE;
		IF NOT fbSoEWritePassword.Busy AND NOT fbSoEWritePassword.Error THEN
			iStep							:= iStep + 10;
		ELSIF fbSoEWritePassword.Error THEN
			udiErrorID						:= fbSoEWritePassword.AdsErrId;
			uiSoEErrorID					:= fbSoEWritePassword.SercosErrId;
			iLastStep						:= iStep;
			iStep							:= 999;
		END_IF
	
	110:															// Ignore offset error (P-0-0278), channel 1	
		P_0_0278_Value						:= 1;
		fbSoEWrite_ByDriveRef.stDriveRef	:= stDriveRef;
		fbSoEWrite_ByDriveRef.stDriveRef.nDriveNo:= 0;
		fbSoEWrite_ByDriveRef.nIdn			:= P_0_IDN + 278;		// SoE Parameters Group P-0-IDN offset
		fbSoEWrite_ByDriveRef.nElement		:= EC_SOE_ELEMENT_VALUE;// Change value of the parameter
		fbSoEWrite_ByDriveRef.pSrcBuf		:= ADR(P_0_0278_Value);
		fbSoEWrite_ByDriveRef.cbBufLen		:= SIZEOF(P_0_0278_Value);
		fbSoEWrite_ByDriveRef.bExecute		:= TRUE;
		iStep								:= iStep + 10;				
		
	120,160:														// Writing done ?		
		fbSoEWrite_ByDriveRef.bExecute		:= FALSE;
		IF NOT fbSoEWrite_ByDriveRef.bBusy AND NOT fbSoEWrite_ByDriveRef.bError THEN
			iStep							:= iStep + 10;
		ELSIF fbSoEWrite_ByDriveRef.bError THEN
			udiErrorID						:= fbSoEWrite_ByDriveRef.iAdsErrId;
			uiSoEErrorID					:= fbSoEWrite_ByDriveRef.iSercosErrId;
			iLastStep						:= iStep;
			iStep							:= 999;
		END_IF	
		
	130:															// reset second channel if needed
		fbSoERead_ByDriveRef.stDriveRef		:= stDriveRef;
		fbSoERead_ByDriveRef.nIdn			:= P_0_IDN + 324;		// SoE Parameters Group P-0-IDN offset
		fbSoERead_ByDriveRef.nElement		:= EC_SOE_ELEMENT_VALUE;// Change value of the parameter
		fbSoERead_ByDriveRef.pDstBuf		:= ADR(stSoE_String);
		fbSoERead_ByDriveRef.cbBufLen		:= SIZEOF(stSoE_String);
		fbSoERead_ByDriveRef.bExecute		:= TRUE;
		iStep								:= iStep + 10;				
		
	140:															// Reading done ?	skip reseting channel 2 for AX51xx	
		fbSoERead_ByDriveRef.bExecute		:= FALSE;
		IF NOT fbSoERead_ByDriveRef.bBusy AND NOT fbSoERead_ByDriveRef.bError THEN
			bDualChannel := STRING_TO_BYTE(MID(stSoE_String.strData, 1, 4)) = 2;		// Sprawdza nazwe AX5xxx i rozpoznaje ilosc kanalow
			IF bDualChannel THEN
				iStep						:= iStep + 10;			// reset channel 2
			ELSE
				iStep						:= iStep + 30;			// skip reseting channel 2
			END_IF
		ELSIF fbSoERead_ByDriveRef.bError THEN
			udiErrorID						:= fbSoERead_ByDriveRef.iAdsErrId;
			uiSoEErrorID					:= fbSoERead_ByDriveRef.iSercosErrId;
			iLastStep						:= iStep;
			iStep							:= 999;
		END_IF	

	150:															// Ignore offset error (P-0-0278), channel 2
		fbSoEWrite_ByDriveRef.stDriveRef.nDriveNo:= 1;
		fbSoEWrite_ByDriveRef.bExecute		:= TRUE;
		iStep								:= iStep + 10;

	170:															// Reset Drive (S-0-0099)
		fbSoEReset.Execute					:= TRUE; 
		fbSoEReset.NetId					:= ''; 
		iStep								:= iStep + 10;
		
	180:															// Wait for drive reset (S-0-0099)
		fbSoEReset.Execute					:= FALSE;
		IF NOT fbSoEReset.Busy AND NOT fbSoEReset.Error THEN
			iStep							:= iStep + 10;
		ELSIF fbSoEReset.Error THEN
			udiErrorID						:= fbSoEReset.AdsErrId;
			uiSoEErrorID					:= fbSoEReset.SercosErrId;
			iLastStep						:= iStep;
			iStep							:= 999;
		END_IF

	190:															// Request OP State
		fbChangeSlaveState.byReguestedState	:= EC_DEVICE_STATE_OP;
		fbChangeSlaveState.bExecute			:= TRUE;
		iStep								:= iStep+10;
	
	200:															// Wait till state changed
		fbChangeSlaveState.bExecute			:= FALSE;	
		IF NOT fbChangeSlaveState.bBusy AND NOT fbChangeSlaveState.bError THEN
			iStep							:= iStep + 10;
		ELSIF NOT fbChangeSlaveState.bBusy AND fbChangeSlaveState.bError THEN
			udiErrorID						:= fbChangeSlaveState.udiErrorID;
			iLastStep						:= iStep;
			iStep 							:= 999;
		END_IF				

	210:															// Set new encoder offset	
		fbSoEAX5000SetPositionOffset.Feedback:= ePositionOffsetFeedback1;	// set to feedback 1 only
		fbSoEAX5000SetPositionOffset.Execute:= TRUE; 
		iStep								:= iStep + 10;

	220:															//	offset set already?
		fbSoEAX5000SetPositionOffset.Execute:= FALSE;
		IF NOT fbSoEAX5000SetPositionOffset.Busy AND NOT fbSoEAX5000SetPositionOffset.Error THEN
			iStep							:= iStep + 10;
		ELSIF fbSoEAX5000SetPositionOffset.Error THEN
			udiErrorID						:= fbSoEAX5000SetPositionOffset.ErrorID;
			iLastStep						:= iStep;
			iStep							:= 999;
		END_IF
	
	230:															//	FB Termination
		bBusy								:= FALSE;
		iStep								:= 0;

	999:															//	ERROR State
		bBusy								:=	FALSE;
		bError								:=	TRUE;
		iStep								:=	0;
	
END_CASE

fbAdsRead();
fbChangeSlaveState();
fbSoEWritePassword(Axis:=Axis);
fbSoEAX5000SetPositionOffset(Axis:=Axis);
fbSoEReadDiagNumber(Axis:=Axis);
fbSoEReset(Axis:=Axis);
fbSoEWrite_ByDriveRef();
fbSoERead_ByDriveRef();

END_FUNCTION_BLOCK

// ---- POUs/Programy/Hbot/AxisOnline/POUsAxisOnline/AX5000/FB_ChangeEtherCATSlaveState.TcPOU
//==================================================================================================
//							Beckhoff Automation Poland
//									23.05.2018
//	Blok zmienia stan EtherCAT Slave i monitoruje flage ukonczenia
//
//	Niezbedne biblioteki: Tc2_EtherCAT
//
// 	v1.1	|| TC v 3.1.4022.16	|| - optymalizacja kodu
// 	v1.0	|| TC v 3.1.4020.32	|| - pierwsza wersja
//==================================================================================================
FUNCTION_BLOCK FB_ChangeEtherCATSlaveState
VAR_INPUT
	bExecute								: BOOL;							// Start on rising edge
	sEtherCAT_NetID							: STRING;						// EtherCAT Master NetID
	nSlaveAddr								: UINT;							// EtherCAT Drive slave port
	byReguestedState						: BYTE;							(* 	16#1- EC_DEVICE_STATE_INIT  
																				16#2- EC_DEVICE_STATE_PREOP     
																				16#3- EC_DEVICE_STATE_BOOTSTRAP     
																				16#4- EC_DEVICE_STATE_SAFEOP  
																				16#8- EC_DEVICE_STATE_OP
																				16#10- EC_DEVICE_STATE_ERROR  *)
END_VAR
VAR_OUTPUT
	byActualState							: BYTE;							(* 	16#1-EC_DEVICE_STATE_INIT  
																				16#2-EC_DEVICE_STATE_PREOP     
																				16#3-EC_DEVICE_STATE_BOOTSTRAP     
																				16#4-EC_DEVICE_STATE_SAFEOP  
																				16#8-EC_DEVICE_STATE_OP
																				16#10-EC_DEVICE_STATE_ERROR  *)
	bBusy									: BOOL;
	bDone									: BOOL;
	bError									: BOOL;
	udiErrorID								: UDINT;	
END_VAR
VAR	
	fbEcReqSlaveState						: FB_EcReqSlaveState;
	fbEcGetSlaveState						: FB_EcGetSlaveState;
	timerTON								: TON;
	rtExecute								: R_TRIG;
	iState									: INT;
	iTry									: INT;							// number of tries
END_VAR

timerTON(PT:=T#500MS);
rtExecute(CLK:=bExecute);

CASE iState OF

	0:																// Init parameters
		IF rtExecute.Q THEN
			bBusy							:= TRUE;
			bDone							:= FALSE;
			bError							:= FALSE;
			udiErrorID						:= 0;
			iTry							:= 0;
			fbEcReqSlaveState.sNetId		:= sEtherCat_NetID; 
			fbEcGetSlaveState.sNetId		:= sEtherCat_NetID; 
			fbEcReqSlaveState.nSlaveAddr	:= nSlaveAddr; 
			fbEcGetSlaveState.nSlaveAddr	:= nSlaveAddr;
			fbEcReqSlaveState.state			:= byReguestedState;
			fbEcReqSlaveState.bExecute		:= TRUE;
			iState							:= iState + 10;			
		END_IF
		
	10:																// State request
		fbEcReqSlaveState.bExecute			:= FALSE;
		IF NOT fbEcReqSlaveState.bBusy THEN
			IF fbEcReqSlaveState.bError THEN
				iState						:= 99;
			ELSE
				iState						:= iState + 10;
			END_IF
		END_IF

		
	20:																// Request every 0.5s
		timerTON.IN							:= TRUE;
		IF timerTON.Q THEN
			timerTON.IN						:= FALSE;
			fbEcGetSlaveState.bExecute		:= TRUE;
			iState							:= iState + 10;
		END_IF
		
	30:																// Done already?
		fbEcGetSlaveState.bExecute			:= FALSE;	
		IF NOT fbEcGetSlaveState.bBusy THEN
			IF NOT fbEcGetSlaveState.bError AND fbEcGetSlaveState.state.deviceState = fbEcReqSlaveState.state THEN
				bBusy						:= FALSE;
				bDone						:= TRUE;
				iState						:= 0;
			ELSIF iTry = 40 THEN
				iState						:= 99;
			ELSE
				iTry						:= iTry + 1;
				iState						:= iState - 10;			
			END_IF
			byActualState					:= fbEcGetSlaveState.state.deviceState;
		END_IF
		
	99:																// ERROR STATE
		bError 								:= TRUE;
		bBusy								:= FALSE;
		udiErrorID							:= fbEcReqSlaveState.nErrId + fbEcGetSlaveState.nErrId;
		iState								:= 0;
		
END_CASE

fbEcReqSlaveState();
fbEcGetSlaveState();

END_FUNCTION_BLOCK

// ---- POUs/Programy/Hbot/AxisOnline/POUsAxisOnline/AX5000/FB_MotorMonitoringAX5000.TcPOU
//==================================================================================================
//							Beckhoff Automation Poland
//									23.05.2018
//	Blok funkcyjny pozwala na monitorowanie i ograniczanie momentu oraz monitoring parametru I2T dla AX5xxx.
//	Zmienne do zlinkowania zadeklarowane są wewnątrz bloku.
//	Ograniczenie i monitorowanie momentu
//	Ograniczenie momentu podawane jest przez wejście rTorqueLimit.
//	Na wyjściu podana jest wartość surowa w %, jak i przeskalowana na A (prąd) i Nm (moment).
//	Blok zwraca wartości bieżące, przefiltrowane i maksymalne.
//	Wartości maksymalne mogą być wyzerowane za pomocą zmiennej bReset.
//	Wewnętrznie wykorzystany jest blok FB_FilterEx.
//	I2T: 	Określamy okno czasowe pomiaru
//
// 	v1.1	|| TC v 3.1.4022.16		|| - optymalizacja kodu
//  v1.0	|| TC v 3.1.4022.16		|| bazuje na FB_TorqueMonitoringEx2, dodane wyjscia zgodne z blokiem do AX8000 
//==================================================================================================
FUNCTION_BLOCK FB_MotorMonitoringAX5000
VAR CONSTANT
	rTorqueLimitLow					: REAL 		:= 0.01;				// Low limit used for bipolar torque limit value
	rTorqueLimitHigh				: REAL		:= 100.0;				// High limit used for bipolar torque limit value
END_VAR
VAR_INPUT
	bReset							: BOOL;
	rTorqueLimit					: REAL 		:= rTorqueLimitHigh; 	// Bipolar torque limit: 0-500%, resolution 0.1%, value goes to: 16#6072 (Ch A)/ 16#6872 (Ch B)
	tI2T_Window						: TIME 		:= T#1M;
END_VAR
VAR_OUTPUT
	bError							: BOOL; 							// Communication error *)
	iAdsErrId						: UINT;								// Forwarded output FB_SoeRead
	iSercosErrId					: UINT;								// Forwarded output FB_SoeRead
	bInitialized					: BOOL;								// TRUE - Motor data read without errors, so it's possible to calculate torqe and current values in metric units
	bWarning						: BOOL;								// Overcurrent (rCurrentF > rRatedCurrent)
	rWarningCurrent					: REAL; 							// P_0_0093_Value in [A]
	rTorquePerc						: REAL;								// [%]
	rTorquePercMax					: REAL;								// Max [%]	
	rTorque							: REAL; 							// [Nm]
	rTorqueF						: REAL;								// Filtered
	rTorqueMax						: REAL;								// Max
	rCurrent						: REAL; 							// [A]
	rCurrentF						: REAL;								// Filtered
	rCurrentMax						: REAL;								// Max
	rI2T							: REAL; 							// % nominal
	rI2TMax							: REAL;
END_VAR
VAR_IN_OUT
	Axis							: AXIS_REF;
END_VAR
VAR
	fbSoERead						: FB_SoeRead;
	iStep							: INT;
	arr_S_0_0030_Value				: ARRAY [1..66] OF BYTE;
	S_0_0030_Value					: STRING;
	bDriveFirmware_2_10				: BOOL;
	P_0_0092_Value					: DWORD;
	P_0_0093_Value					: DWORD;
	P_0_0070_Value					: DWORD;
	S_0_0111_Value					: DWORD;
	uiBipolarTorqueLimitValue AT %Q*	: UINT; 								// Raw data, linked to Bipolar torque limit value MDT, S-0-0092
	iTorque 							: INT; 								// -1000 .. 1000 - RAW values the same as process image
	rTorqueRAW						: REAL; 							// -1000 .. 1000 - RAW values the same as process image	
	rPeakCurrent					: REAL; 							// P_0_0092_Value in [A]
	rFactor							: REAL; 							// iTorque -1000..1000 --> - rPeakCurrent .. rPeakCurrent
	rContinuousStallTorque			: REAL; 							// P_0_0070_Value [Nm]
	rContinuousStallCurrent			: REAL; 							// S_0_0111_Value [A]
	rTorqueConstant					: REAL; 							// P_0_0070_Value/S_0_0111_Value [Nm/A]
	fbFilterEx						: FB_FilterEx;

	rI2T_pom						: REAL 		:= 0.0;
	rI2T_Window						: REAL;
	bFlag_1							: BOOL 		:= FALSE;
	iCycles							: INT;
	rCycleTime_pom					: REAL;
	iCounter						: INT;
	rBuffer							: ARRAY[1..100] OF REAL;
	rBuffer_2						: ARRAY[1..100] OF REAL;

	rCycleTime						: REAL;								// Ustawiony czas Tasku w ms
	fbGETCURTASKINDEX   			: GETCURTASKINDEX;					// Blok sprawdzajcy numer Tasku
	BIndex							: BYTE;								// Nr Tasku
	tonReset						: TON;
END_VAR

CASE iStep OF
	0: (*Init*)
		bError 						:= FALSE;
		bInitialized				:= FALSE;
		iAdsErrId 					:= 0;
		iSercosErrId				:= 0;
		iStep 						:= iStep + 10;
	
	10: (* Read S_0_0030 *)
		fbSoERead.Idn 				:= S_0_IDN + 30;
		fbSoERead.Element			:= EC_SOE_ELEMENT_VALUE;
		fbSoERead.pDstBuf			:= ADR(arr_S_0_0030_Value);
		fbSoERead.BufLen			:= SIZEOF(arr_S_0_0030_Value);
		fbSoERead.Execute			:= TRUE;
		iStep 						:= iStep + 10;
	
	20:	(* Read Drive firmware version *)
		IF NOT fbSoERead.Busy AND NOT fbSoERead.Error THEN
			fbSoERead.Execute		:= FALSE;
			S_0_0030_Value			:= '';																// Set emtpy string for save data
			FOR iCounter := 1 TO 	UINT_TO_BYTE(SIZEOF(arr_S_0_0030_Value)) 	DO
				S_0_0030_Value		:= CONCAT(S_0_0030_Value, F_ToCHR(arr_S_0_0030_Value[iCounter]));	// Translate ASCII to string 
			END_FOR
			bDriveFirmware_2_10 	:= INT_TO_BOOL(FIND(S_0_0030_Value,'Firmware: v2.10'));				// Check if firmware 2.10 / 2.06
			iStep 					:= iStep + 10;
		END_IF
		IF fbSoERead.Error THEN
			iStep 					:= 500;
		END_IF

	30: (*Read P_0_0092*)
		fbSoERead.Idn 				:= P_0_IDN + 92;
		fbSoERead.Element			:= EC_SOE_ELEMENT_VALUE;
		fbSoERead.pDstBuf			:= ADR(P_0_0092_Value);
		fbSoERead.BufLen			:= SIZEOF(P_0_0092_Value);
		fbSoERead.Execute			:= TRUE;
		iStep 						:= iStep + 10;

	40:
		IF NOT fbSoERead.Busy AND NOT fbSoERead.Error THEN
			rPeakCurrent 			:= DWORD_TO_REAL(P_0_0092_Value)/1000.0;
			rFactor 				:= DWORD_TO_REAL(P_0_0092_Value)/1000000.0;
			fbSoERead.Execute		:= FALSE;
			iStep 					:= iStep + 10;
		END_IF
		IF fbSoERead.Error THEN
			iStep 					:= 500;
		END_IF
		
	50:
		(*Read P_0_0070*)	
		fbSoERead.Idn 				:= P_0_IDN + 70;
		fbSoERead.Element			:= EC_SOE_ELEMENT_VALUE; 
		fbSoERead.pDstBuf			:= ADR(P_0_0070_Value);
		IF bDriveFirmware_2_10 THEN
			fbSoERead.BufLen		:= 4;
		ELSE
			fbSoERead.BufLen		:= 2;
		END_IF
		fbSoERead.Execute			:= TRUE;
		iStep 						:= iStep + 10;

	60:
		IF NOT fbSoERead.Busy AND NOT fbSoERead.Error THEN
			rContinuousStallTorque 	:= DWORD_TO_REAL(P_0_0070_Value)/100;
			fbSoERead.Execute		:= FALSE;
			iStep 					:= iStep + 10;
		END_IF
		IF fbSoERead.Error OR P_0_0070_Value = 0 THEN
			iStep 					:= 500;
		END_IF

	70: (* Read S_0_0111*)
		fbSoERead.Idn 				:= S_0_IDN + 111;
		fbSoERead.Element			:= EC_SOE_ELEMENT_VALUE;
		fbSoERead.pDstBuf			:= ADR(S_0_0111_Value);
		fbSoERead.BufLen			:= SIZEOF(S_0_0111_Value);
		fbSoERead.Execute			:= TRUE;
		iStep 						:= iStep + 10;

	80:
		IF NOT fbSoERead.Busy AND NOT fbSoERead.Error THEN
			IF S_0_0111_Value <> 0 THEN
				rContinuousStallCurrent := DWORD_TO_REAL(S_0_0111_Value)/1000;
				rTorqueConstant 	:= rContinuousStallTorque/rContinuousStallCurrent;
				fbSoERead.Execute	:= FALSE;
				iStep 				:= iStep + 10;
			ELSE
				iStep				:= 500;
			END_IF
		END_IF
		IF fbSoERead.Error THEN
			iStep 					:= 500;
		END_IF

	90: (* Read P_0_0093*)
		fbSoERead.Idn 				:= P_0_IDN + 93;
		fbSoERead.Element			:= EC_SOE_ELEMENT_VALUE;
		fbSoERead.pDstBuf			:= ADR(P_0_0093_Value);
		fbSoERead.BufLen			:= SIZEOF(P_0_0093_Value);
		fbSoERead.Execute			:= TRUE;
		iStep 						:= iStep + 10;

	100:
		IF NOT fbSoERead.Busy AND NOT fbSoERead.Error THEN
			rWarningCurrent 			:= DWORD_TO_REAL(P_0_0093_Value)/1000;
			fbSoERead.Execute		:= FALSE;
			iStep 					:= iStep + 10;
		END_IF
		IF fbSoERead.Error THEN
			bInitialized			:= TRUE;
			iStep 					:= 500;
		END_IF

	110: (*Calculations*)
		rCurrent 					:= rTorqueRAW * rFactor;
		rTorque 					:= rCurrent * rTorqueConstant;

	500: (* Error Case *)
		iStep 						:= 0;
		fbSoERead(Execute:= FALSE,Axis:= Axis);
		bError 						:= TRUE;
		iAdsErrId 					:= fbSoERead.AdsErrId;
		iSercosErrId				:= fbSoERead.SercosErrId;
		tonReset(IN:= TRUE, PT:= T#1S);
		IF tonReset.Q THEN
			tonReset(IN:= FALSE);
		END_IF
END_CASE
//===================== Limit output torque =====================
IF rTorqueLimit < rTorqueLimitLow THEN
	uiBipolarTorqueLimitValue 			:= REAL_TO_UINT(rTorqueLimitHigh);			// Secure against 0 value - probably empty var connected to input
ELSE
	uiBipolarTorqueLimitValue 			:= REAL_TO_UINT(LIMIT(rTorqueLimitLow,rTorqueLimit,rTorqueLimitHigh))*10;
END_IF

//=============== Read cycle time ===============
fbGETCURTASKINDEX(index => BIndex);
rCycleTime := UDINT_TO_REAL(_TaskInfo[BIndex].CycleTime)/10000.0;

//=============== Calculate algorithm sampling time ===============
rI2T_Window := TIME_TO_REAL(tI2T_Window);
rCycleTime_pom := rI2T_Window/100 ;

IF rCycleTime_pom < rCycleTime THEN
	rCycleTime_pom := rCycleTime;
END_IF

//=============== Filter current value ===============
fbFilterEx(rIn:= rCurrent, tTimeConstant:= REAL_TO_TIME(rCycleTime_pom), rOut=> rCurrentF);
rTorqueF := rCurrentF * rTorqueConstant;

//=============== Save torque and current max values ===============
IF ABS(rCurrentMax) < ABS(rCurrentF) THEN
	rTorquePercMax						:= rTorquePerc;
	rCurrentMax 						:= rCurrentF;
	rTorqueMax							:= rTorqueF;
END_IF
//======================== Set outputs ==========================
rTorquePerc								:= LREAL_TO_REAL(Axis.NcToPlc.ActTorque); 		// [%]
rTorqueRAW 								:= rTorquePerc*10;								// -1000 .. 1000 - RAW values the same as process image


//=============== Oblicznie I2T ===============
//======== b_Flag_1 is set to TRUE when PLC cycle matches with algorythm sampling rate ========

IF rCycleTime <> 0 THEN
	IF iCycles < rCycleTime_pom/rCycleTime  THEN
		iCycles := iCycles + 1;
		bFlag_1 := FALSE;
	ELSE
		iCycles := 0;
		bFlag_1 := TRUE;
	END_IF
END_IF

(*Save momentary I2T values in ring buffer*)

IF bFlag_1 THEN
	FOR iCounter :=1 TO 99 DO
		rBuffer[iCounter] := rBuffer[iCounter+1];
		rBuffer_2[iCounter] := rBuffer_2[iCounter+1];
	END_FOR
	rBuffer[100] := rCurrentF *rCurrentF* rCycleTime_pom;
	rBuffer_2[100] := rWarningCurrent *rWarningCurrent* rCycleTime_pom;
END_IF

rI2T := 0;
rI2T_pom := 0;

(*Calculate I2T parameter*)

FOR iCounter:=1 TO 100 BY 1 DO
	rI2T := rI2T + rBuffer[iCounter];
	rI2T_pom := rI2T_pom + rBuffer_2[iCounter];
END_FOR

(*Scale I2T to 0-100% range*)

IF rI2T_pom  <> 0  THEN
	rI2T := rI2T/rI2T_pom*100;
END_IF

IF rI2TMax < rI2T THEN
	rI2TMax := rI2T;
END_IF

// Flaga Overcurrent (rCurrentF > rRatedCurrent)
bWarning := rCurrentF > rWarningCurrent;

IF bReset THEN
	rCurrentMax := 0;
	rTorqueMax := 0;
	rI2TMax := 0;
	FOR iCounter:=1 TO 100 BY 1 DO
		rBuffer[iCounter] := 0;
		rBuffer_2[iCounter] := 0;
	END_FOR;
END_IF

//========= Wywolanie bloku odczytu =========
fbSoERead(
	NetId:= '',
	Timeout:= T#1s,
	Axis:= Axis);

END_FUNCTION_BLOCK

// ---- POUs/Programy/Hbot/AxisOnline/POUsAxisOnline/FBs/FB_FilterEx.TcPOU
//==================================================================================================
//							Beckhoff Automation Poland
//									23.11.2016
//			Bloczek do filtru inercyjnego do wygladzania przebiegow,					
//					czas próbkowania wyliczany wewnętrznie
//  v1.1	|| TC v 3.1.4020.28		|| - poprawienie inicjalizacji, notacja wegierska
// 	v1.0	|| TC v 3.1.4020.0		|| - pierwsza wersja
//==================================================================================================
FUNCTION_BLOCK FB_FilterEx
VAR_INPUT
	rIn										: REAL;					// Sygnal wejsciowy
	tTimeConstant							: TIME;					// Stala czasowa T gdy rOut = 0,63 * rIn 
END_VAR
VAR_OUTPUT
	rOut									: REAL;					// Przefiltrowany sygnal wyjsciowy, 
END_VAR
VAR
	rLastOut								: REAL;					// Wartosc wyjscia w poprzednim cyklu
	rCycleTime								: REAL; 				// [ms]
	rTimeConst								: REAL;					// [ms]
	tX										: TIME;					// Aktualny czas
	tY 										: TIME;					// Zmienna pomocnicza, poprzedni czas
	tCycleTime								: TIME;					// Wyliczony czas cyklu
	bFirstCycle								: BOOL := TRUE;			// Flaga pierwszego cyklu - nie mamy jeszce wyliczonego prawidlowo czasu cylu 
																	// - potrzebujemy dwoch cylki do odjecia czasu
END_VAR

// Obliczenie czasu cyklu do inkrementu
tX 					:= TIME();
IF NOT bFirstCycle THEN
	tCycleTime 		:= tX - tY;
END_IF
tY 					:= tX;
// Przeliczenie czasu na typ REAL
rCycleTime 			:= TIME_TO_REAL(tCycleTime);
rTimeConst 			:= TIME_TO_REAL(tTimeConstant);
// Wyliczenie wyjscia tylko jesli stala czasowa wieksza od 1 ms i zakonczylismy inicjalizacje
IF NOT bFirstCycle AND rTimeConst > 0.001 THEN
	rOut 			:= rLastOut + (rIn - rLastOut) * rCycleTime/rTimeConst;
	rLastOut 		:= rOut;
END_IF
// Zerowanie flagu pierwszego cyklu
bFirstCycle 		:= FALSE;

END_FUNCTION_BLOCK

// ---- POUs/Programy/Hbot/AxisOnline/POUsAxisOnline/AX5000/FB_HoldingBrakeCtrlAX5000.TcPOU
//==================================================================================================
//							Beckhoff Automation Poland
//									23.05.2018
//	Blok funkcyjny kontroli luzownika w silniku podpietym do AX5000. Przewaga ForceLock
//	Datatype:		ENUM (INT16)
//	Enum Value:		0 (0x00): 	Release_force
//					1 (0x01): 	Force_lock
//					2 (0x02): 	Force_unlock
//
// 	v1.1	|| TC v 3.1.4022.16	|| - optymalizacja kodu
//  v1.0	|| TC v 3.1.4022.16	|| - pierwsza wersja
//==================================================================================================
FUNCTION_BLOCK FB_HoldingBrakeCtrlAX5000
VAR_INPUT
	bForceLock 						: BOOL;								// 
	bForceUnlock					: BOOL;								// 
END_VAR
VAR_OUTPUT
	bBusy							: BOOL;
	bError							: BOOL; 							// General error: parameter or CoE read.
																		// If bError = TRUE and bInitialized = FALSE - error during read motor data.
																		// If bError = TRUE and bInitialized = TRUE and (iAdsErrId <> 0 or iCANopenErrId <> 0) then I2T read error
																		// If bError = TRUE and bInitialized = TRUE and iAdsErrId = 0 and iCANopenErrId = 0 then parameter error: rTorqueLimit outside permitted range rTorqueLimitLow..rTorqueLimitHigh or Empty stDriveRef
	iAdsErrId						: UINT;								// Forwarded output FB_SoEWrite
	iSecErrId						: UINT;								// Forwarded output FB_SoEWrite
END_VAR
VAR_IN_OUT
	Axis							: AXIS_REF;
END_VAR
VAR
	bExecute						: BOOL;
	iMotorBrakeForce				: INT;								// 0 - Release_force, 1 - Force_lock, 2 - Force_unlock
	fbSoEWrite						: FB_SoEWrite;
	rtForceLock						: R_TRIG;
	rtForceUnlock					: R_TRIG;
	ftForceLock						: F_TRIG;
	ftForceUnlock					: F_TRIG;
END_VAR

{region "Call triggers"}
//======================= Call triggers =========================
rtForceLock(CLK:= bForceLock);
ftForceLock(CLK:= bForceLock);
rtForceUnlock(CLK:= bForceUnlock);
ftForceUnlock(CLK:= bForceUnlock);
bExecute								:= rtForceLock.Q OR ftForceLock.Q OR rtForceUnlock.Q OR ftForceUnlock.Q;
//===============================================================
{endregion}
{region "Main code"}
//========================= Main code ===========================
IF bExecute THEN
	iMotorBrakeForce 						:= 0;										// Clear value
	iMotorBrakeForce.1 						:= bForceUnlock;							// Set force unlock bit
	iMotorBrakeForce 						:= SEL(bForceLock, iMotorBrakeForce, 1);	// Set force lock bit, it has higher priority than unlock
END_IF
	 
fbSoEWrite(
	NetId			:= '' , 
	Idn				:= P_0_IDN + 96 , 
	Element			:= 16#40 , 
	pSrcBuf			:= ADR(iMotorBrakeForce), 
	BufLen			:= SIZEOF(iMotorBrakeForce) , 
	Execute			:= bExecute , 
	Timeout			:= T#2S, 
	Axis			:= Axis , 
	Busy			=> bBusy , 
	Error			=> bError, 
	AdsErrId		=> iAdsErrId, 
	SercosErrId		=> iSecErrId );
//===============================================================
{endregion}

END_FUNCTION_BLOCK

// ---- POUs/Programy/Hbot/AxisOnline/POUsAxisOnline/FBs/FB_NcSWLimitSwitchCtrl.TcPOU
//==================================================================================================
//					Beckhoff Automation Poland
//							23.05.2018
//		Blok funkcyjny zmieniajacy krancowki SW gorna i dolna
// 	v1.2	|| TC v 3.1.4022.16		|| - optymalizacja kodu
// 	v1.1 	|| TC v 3.1.4022.2	 	|| - dodane komentarze do zmiennych
// 	v1.0 	|| TC v 3.1.4020.32 	|| - pierwsza wersja
//==================================================================================================
FUNCTION_BLOCK FB_NcSWLimitSwitchCtrl
VAR_INPUT
	udiAxisID				: UDINT;					// ID osi
	bRead					: BOOL;						// Read SW limit switches values and states
	bWrite					: BOOL;						// Write SW limit switches values and states
	bReset					: BOOL; 					// Not yet
// Set values
	lrSetMinPos				: LREAL;					// SW limit switch minimum
	lrSetMaxPos				: LREAL;					// SW limit switch maximum
	bSetMinMon				: BOOL;						// Enable SW limit switch minimum monitoring
	bSetMaxMon				: BOOL;						// Enable SW limit switch maximum monitoring
END_VAR
VAR_OUTPUT
	//	
	bBusy					: BOOL;						// Read/Write busy
	bError					: BOOL;						// Read/Write error
	udiErrorID				: UDINT;					// Read/Write error ID
// Actual values	
	lrActMinPos				: LREAL;					// Actual SW limit switch minimum
	lrActMaxPos				: LREAL;					// Actual SW limit switch maximum
	bActMinMon				: BOOL;						// SW limit switch minimum monitoring state
	bActMaxMon				: BOOL;						// SW limit switch maximum monitoring state
END_VAR
VAR
	iStepWrite				: INT;
	iStepRead				: INT;
	wSetMinMon				: WORD;
	wSetMaxMon				: WORD;
	wActMinMon				: WORD;
	wActMaxMon				: WORD;
// FBs
	rtRead					: R_TRIG;
	rtWrite					: R_TRIG;
	fbADSREAD				: ADSREAD;
	fbADSWRITE				: ADSWRITE;
END_VAR
VAR CONSTANT
	udiIDXGRP_OFFS			: UDINT := 16#0000_5000;
END_VAR

// Triggery
rtRead(CLK:= bRead, Q=> );
rtWrite(CLK:= bWrite, Q=> );

ACT_ReadParams();
ACT_WriteParams();	

	
// Read parameters
	fbADSREAD(	NETID:= '', 
				PORT:= 500,
				IDXGRP:= udiIDXGRP_OFFS + udiAxisID);
	
// Write parameters
	fbADSWRITE(	NETID:= '', 
				PORT:= 500,
				IDXGRP:= udiIDXGRP_OFFS + udiAxisID);

ACTION ACT_ReadParams:
CASE iStepRead OF

0: // Idle
	IF rtRead.Q AND NOT bBusy THEN
		bBusy 					:= TRUE;
		bError 					:= FALSE;
		udiErrorID				:= 0;
		// MinMon 16#0000_000B;	// 2B
		fbADSREAD.READ			:= TRUE;
		fbADSREAD.IDXOFFS		:= 16#0000_000B;
		fbADSREAD.LEN			:= 2;
		fbADSREAD.DESTADDR		:= ADR(wActMinMon);
		iStepRead				:= iStepRead + 5;
	END_IF
	
5, 15, 25: // Wait CMD for end
	fbADSREAD.READ				:= FALSE;
	IF NOT fbADSREAD.BUSY AND NOT fbADSREAD.ERR THEN
		iStepRead				:= iStepRead + 5;
	ELSIF fbADSREAD.ERR THEN
		iStepRead				:= 1000;
	END_IF
	
10: // udiIDXOFFS_MinPos		: UDINT := 16#0000_000D;	// 8B
	fbADSREAD.READ				:= TRUE;
	fbADSREAD.IDXOFFS			:= 16#0000_000D;
	fbADSREAD.LEN				:= 8;
	fbADSREAD.DESTADDR			:= ADR(lrActMinPos);
	iStepRead					:= iStepRead + 5;

20: // 	udiIDXOFFS_MaxMon		: UDINT := 16#0000_000C;	// 2B
	fbADSREAD.READ				:= TRUE;
	fbADSREAD.IDXOFFS			:= 16#0000_000C;
	fbADSREAD.LEN				:= 2;
	fbADSREAD.DESTADDR			:= ADR(wActMaxMon);
	iStepRead					:= iStepRead + 5;

30: // 		udiIDXOFFS_MaxPos		: UDINT := 16#0000_000E;	// 8B
	fbADSREAD.READ				:= TRUE;
	fbADSREAD.IDXOFFS			:= 16#0000_000E;
	fbADSREAD.LEN				:= 8;
	fbADSREAD.DESTADDR			:= ADR(lrActMaxPos);
	iStepRead					:= iStepRead + 5;
		
35: // 	End
	fbADSREAD.READ				:= FALSE;
	IF NOT fbADSREAD.BUSY AND NOT fbADSREAD.ERR THEN
		bActMinMon				:= wActMinMon.0;
		bActMaxMon				:= wActMaxMon.0;
		bBusy 					:= FALSE;
		iStepRead				:= 0;
	ELSIF fbADSREAD.ERR THEN
		iStepRead				:= 1000;
	END_IF
	
1000:
	bBusy 						:= FALSE;
	bError 						:= TRUE;
	udiErrorID					:= fbADSREAD.ERRID;
	iStepRead					:= 0;

END_CASE
END_ACTION

ACTION ACT_WriteParams:
CASE iStepWrite OF

